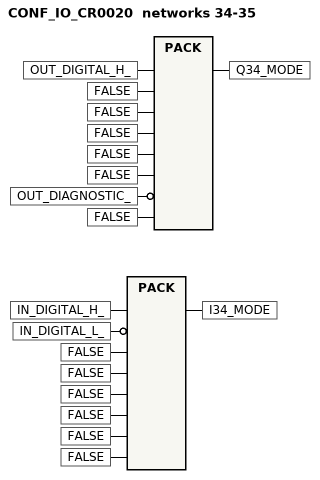
[picture p24: CONF_IO_CR0020 (FBD) networks 34-35]
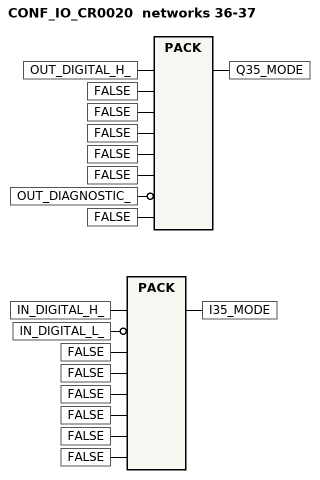
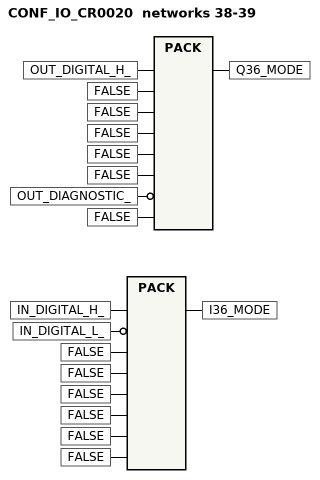
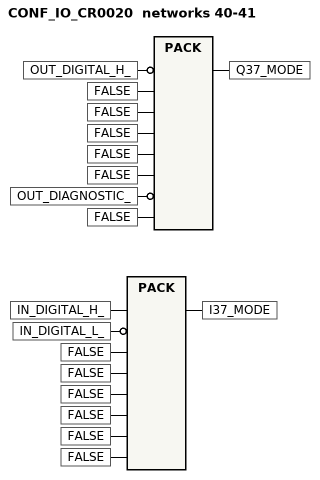
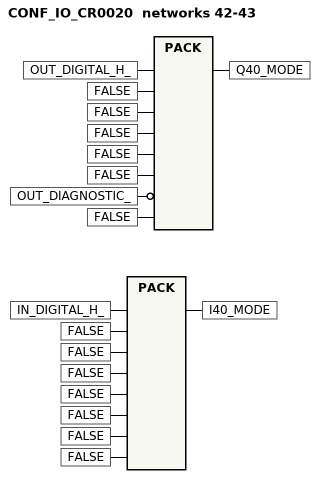
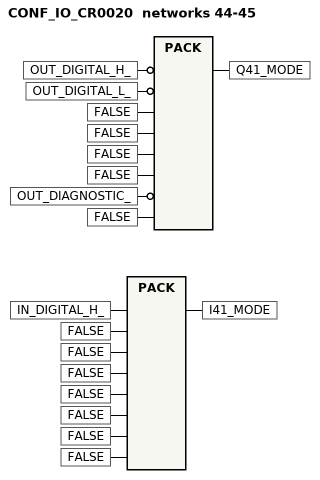
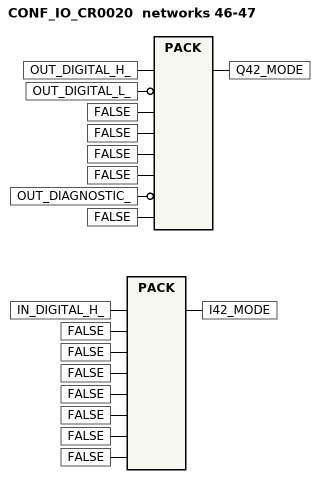
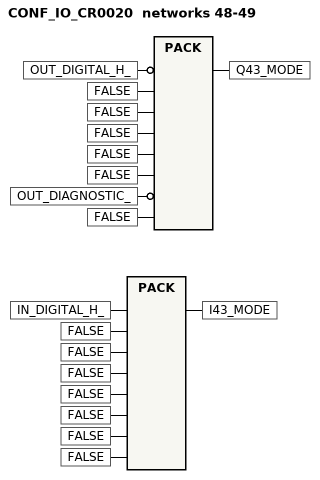
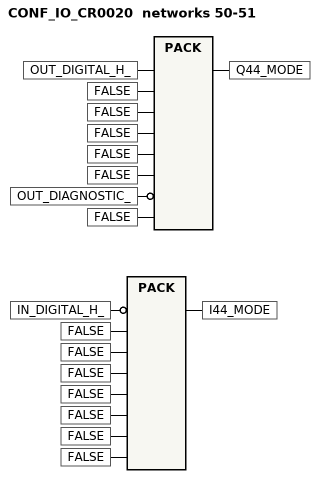
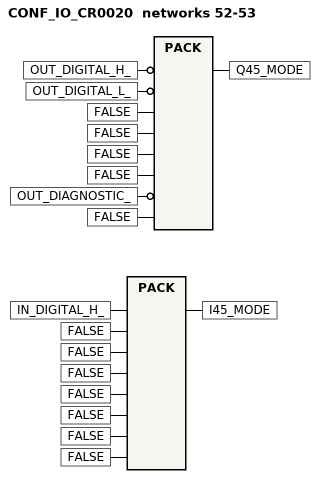
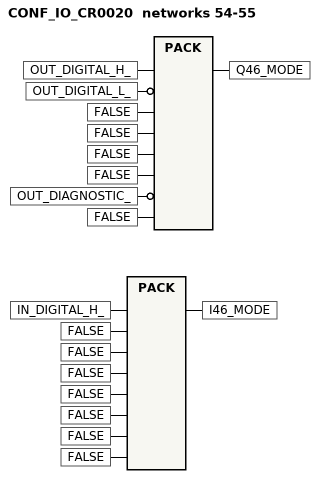
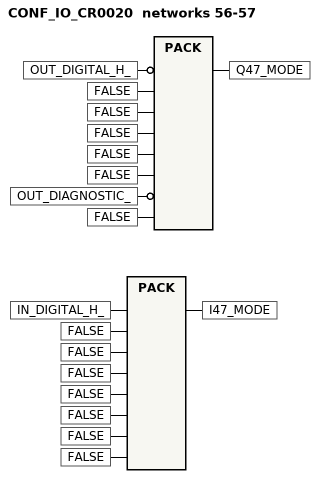
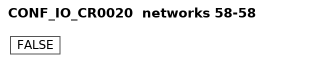
_FBD_ (* Function Block Diagram *)
NETWORK 1
	NOT INIT => >>END
NETWORK 2 (* Configuration byte for analog channel 0 pin 08 Connector 1. No output is connected to this pin. / Default setting:B0:=TRUE,B1:= FALSE,B2:= FALSE,B3:= FALSE,B4:= TRUE,B5:= FALSE,B6:= FALSE,B7:=FALSE *)
	PACK(FALSE, FALSE, IN_CURRENT_, FALSE, FALSE, FALSE, FALSE, FALSE) => I00_MODE
NETWORK 3 (* Configuration byte for analog channel 1 pin 27 Connector 1. No output is connected to this pin. / Default setting:B0:=TRUE,B1:= FALSE,B2:= FALSE,B3:= FALSE,B4:= TRUE,B5:= FALSE,B6:= FALSE,B7:=FALSE *)
	PACK(FALSE, FALSE, IN_CURRENT_, FALSE, FALSE, FALSE, FALSE, FALSE) => I01_MODE
NETWORK 4 (* Configuration byte for analog channel 2 pin 09 Connector 1. No output is connected to this pin. / Default setting:B0:=TRUE,B1:= FALSE,B2:= FALSE,B3:= FALSE,B4:= TRUE,B5:= FALSE,B6:= FALSE,B7:=FALSE *)
	PACK(FALSE, FALSE, IN_CURRENT_, FALSE, FALSE, FALSE, FALSE, FALSE) => I02_MODE
NETWORK 5 (* Configuration byte for analog channel 3 pin 28 Connector 1. No output is connected to this pin. / Default setting:B0:=TRUE,B1:= FALSE,B2:= FALSE,B3:= FALSE,B4:= TRUE,B5:= FALSE,B6:= FALSE,B7:=FALSE *)
	PACK(FALSE, FALSE, IN_CURRENT_, FALSE, FALSE, FALSE, FALSE, FALSE) => I03_MODE
NETWORK 6 (* Configuration byte for analog channel 4 pin 10 Connector 1. No output is connected to this pin. / Default setting:B0:=TRUE,B1:= FALSE,B2:= FALSE,B3:= FALSE,B4:= TRUE,B5:= FALSE,B6:= FALSE,B7:=FALSE *)
	PACK(FALSE, FALSE, IN_CURRENT_, FALSE, FALSE, FALSE, FALSE, FALSE) => I04_MODE
NETWORK 7 (* Configuration byte for analog channel 5 pin 29 Connector 1. No output is connected to this pin. / Default setting:B0:=TRUE,B1:= FALSE,B2:= FALSE,B3:= FALSE,B4:= TRUE,B5:= FALSE,B6:= FALSE,B7:=FALSE *)
	PACK(FALSE, FALSE, IN_CURRENT_, FALSE, FALSE, FALSE, FALSE, FALSE) => I05_MODE
NETWORK 8 (* Configuration byte for analog channel 6 pin 11 Connector 1. No output is connected to this pin. / Default setting:B0:=TRUE,B1:= FALSE,B2:= FALSE,B3:= FALSE,B4:= TRUE,B5:= FALSE,B6:= FALSE,B7:=FALSE *)
	PACK(FALSE, FALSE, IN_CURRENT_, FALSE, FALSE, FALSE, FALSE, FALSE) => I06_MODE
NETWORK 9 (* Configuration byte for analog channel 7 pin 30 Connector 1. No output is connected to this pin. / Default setting:B0:=TRUE,B1:= FALSE,B2:= FALSE,B3:= FALSE,B4:= TRUE,B5:= FALSE,B6:= FALSE,B7:=FALSE *)
	PACK(FALSE, FALSE, IN_CURRENT_, FALSE, FALSE, FALSE, FALSE, FALSE) => I07_MODE
NETWORK 10 (* Configuration byte for input %IX0.12  pin 20 Connector 1. No output is connected to this pin. / Default setting:B0:=TRUE,B1:= FALSE,B2:= FALSE,B3:= FALSE,B4:= FALSE,B5:= FALSE,B6:= FALSE,B7:=FALSE *)
	PACK(IN_DIGITAL_H_, FALSE, FALSE, FALSE, FALSE, FALSE, FALSE, NOT IN_FAST_) => I14_MODE
NETWORK 11 (* Configuration byte for input %IX0.13  pin 02 Connector 1. No output is connected to this pin. / Default setting:B0:=TRUE,B1:= FALSE,B2:= FALSE,B3:= FALSE,B4:= FALSE,B5:= FALSE,B6:= FALSE,B7:=FALSE *)
	PACK(IN_DIGITAL_H_, FALSE, FALSE, FALSE, FALSE, FALSE, FALSE, NOT IN_FAST_) => I15_MODE
NETWORK 12 (* Configuration byte for input %IX0.14  pin 21 Connector 1. No output is connected to this pin. / Default setting:B0:=TRUE,B1:= FALSE,B2:= FALSE,B3:= FALSE,B4:= FALSE,B5:= FALSE,B6:= FALSE,B7:=FALSE *)
	PACK(IN_DIGITAL_H_, FALSE, FALSE, FALSE, FALSE, FALSE, FALSE, IN_FAST_) => I16_MODE
NETWORK 13 (* Configuration byte for input %IX0.15  pin 38 Connector 1. No output is connected to this pin. / Default setting:B0:=TRUE,B1:= FALSE,B2:= FALSE,B3:= FALSE,B4:= FALSE,B5:= FALSE,B6:= FALSE,B7:=FALSE *)
	PACK(IN_DIGITAL_H_, FALSE, FALSE, FALSE, FALSE, FALSE, FALSE, IN_FAST_) => I17_MODE
NETWORK 14 (* Configuration byte for input %IX1.04  pin 19 Connector 1. No output is connected to this pin. / Default setting:B0:=TRUE,B1:= FALSE,B2:= FALSE,B3:= FALSE,B4:= FALSE,B5:= FALSE,B6:= FALSE,B7:=FALSE *)
	PACK(IN_DIGITAL_H_, FALSE, FALSE, FALSE, FALSE, FALSE, FALSE, IN_FAST_) => I24_MODE
NETWORK 15 (* Configuration byte for input %IX1.05  pin 55 Connector 1. No output is connected to this pin. / Default setting:B0:=TRUE,B1:= FALSE,B2:= FALSE,B3:= FALSE,B4:= FALSE,B5:= FALSE,B6:= FALSE,B7:=FALSE *)
	PACK(IN_DIGITAL_H_, FALSE, FALSE, FALSE, FALSE, FALSE, FALSE, IN_FAST_) => I25_MODE
NETWORK 16 (* Configuration byte for input %IX1.06  pin 18 Connector 1. No output is connected to this pin. / Default setting:B0:=TRUE,B1:= FALSE,B2:= FALSE,B3:= FALSE,B4:= FALSE,B5:= FALSE,B6:= FALSE,B7:=FALSE *)
	PACK(IN_DIGITAL_H_, FALSE, FALSE, FALSE, FALSE, FALSE, FALSE, IN_FAST_) => I26_MODE
NETWORK 17 (* Configuration byte for input %IX1.07  pin 37 Connector 1. No output is connected to this pin. / Default setting:B0:=TRUE,B1:= FALSE,B2:= FALSE,B3:= FALSE,B4:= FALSE,B5:= FALSE,B6:= FALSE,B7:=FALSE *)
	PACK(IN_DIGITAL_H_, FALSE, FALSE, FALSE, FALSE, FALSE, FALSE, IN_FAST_) => I27_MODE
NETWORK 18 (* Configuration byte for output %QX0.00  pin 44 Connector 1. The input %IX0.08 on pin 44 has no configuration byte. / Default setting:B0:=TRUE,B1:= FALSE,B2:= FALSE,B3:= FALSE,B4:= FALSE,B5:= FALSE,B6:= FALSE,B7:=TRUE *)
	PACK(OUT_DIGITAL_H_, FALSE, NOT OUT_CURRENT_, FALSE, FALSE, FALSE, NOT OUT_DIAGNOSTIC_, OUT_OVERLOAD_PROTECTION_) => Q10_MODE
NETWORK 19 (* Configuration byte for output %QX0.01  pin 45 Connector 1. The input %IX0.09 on pin 45 has no configuration byte. / Default setting:B0:=TRUE,B1:= FALSE,B2:= FALSE,B3:= FALSE,B4:= FALSE,B5:= FALSE,B6:= FALSE,B7:=TRUE *)
	PACK(OUT_DIGITAL_H_, FALSE, NOT OUT_CURRENT_, FALSE, FALSE, FALSE, NOT OUT_DIAGNOSTIC_, OUT_OVERLOAD_PROTECTION_) => Q11_MODE
NETWORK 20 (* Configuration byte for output %QX0.02  pin 46 Connector 1. The input %IX0.10 on pin 46 has no configuration byte. / Default setting:B0:=TRUE,B1:= FALSE,B2:= FALSE,B3:= FALSE,B4:= FALSE,B5:= FALSE,B6:= FALSE,B7:=TRUE *)
	PACK(OUT_DIGITAL_H_, FALSE, NOT OUT_CURRENT_, FALSE, FALSE, FALSE, NOT OUT_DIAGNOSTIC_, OUT_OVERLOAD_PROTECTION_) => Q12_MODE
NETWORK 21 (* Configuration byte for output %QX0.03  pin 47 Connector 1. The input %IX0.11 on pin 47 has no configuration byte. / Default setting:B0:=TRUE,B1:= FALSE,B2:= FALSE,B3:= FALSE,B4:= FALSE,B5:= FALSE,B6:= FALSE,B7:=TRUE *)
	PACK(OUT_DIGITAL_H_, FALSE, NOT OUT_CURRENT_, FALSE, FALSE, FALSE, NOT OUT_DIAGNOSTIC_, OUT_OVERLOAD_PROTECTION_) => Q13_MODE
NETWORK 22 (* Configuration byte for output %QX0.04  pin 36 Connector 1. The input %IX1.00 on pin 36 has no configuration byte. / Default setting:B0:=TRUE,B1:= FALSE,B2:= FALSE,B3:= FALSE,B4:= FALSE,B5:= FALSE,B6:= FALSE,B7:=TRUE *)
	PACK(OUT_DIGITAL_H_, FALSE, NOT OUT_CURRENT_, FALSE, FALSE, FALSE, NOT OUT_DIAGNOSTIC_, OUT_OVERLOAD_PROTECTION_) => Q20_MODE
NETWORK 23 (* Configuration byte for output %QX0.05  pin 54 Connector 1 The input %IX1.01 on pin 54 has no configuration byte. / Default setting:B0:=TRUE,B1:= FALSE,B2:= FALSE,B3:= FALSE,B4:= FALSE,B5:= FALSE,B6:= FALSE,B7:=TRUE *)
	PACK(OUT_DIGITAL_H_, FALSE, NOT OUT_CURRENT_, FALSE, FALSE, FALSE, NOT OUT_DIAGNOSTIC_, OUT_OVERLOAD_PROTECTION_) => Q21_MODE
NETWORK 24 (* Configuration byte for output %QX0.06  pin 17 Connector 1 The input %IX1.02 on pin 17 has no configuration byte. / Default setting:B0:=TRUE,B1:= FALSE,B2:= FALSE,B3:= FALSE,B4:= FALSE,B5:= FALSE,B6:= FALSE,B7:=TRUE *)
	PACK(NOT OUT_DIGITAL_H_, FALSE, NOT OUT_CURRENT_, FALSE, FALSE, FALSE, NOT OUT_DIAGNOSTIC_, OUT_OVERLOAD_PROTECTION_) => Q22_MODE
NETWORK 25 (* Configuration byte for output %QX0.07  pin 53 Connector 1 The input %IX1.03 on pin 53 has no configuration byte. / Default setting:B0:=TRUE,B1:= FALSE,B2:= FALSE,B3:= FALSE,B4:= FALSE,B5:= FALSE,B6:= FALSE,B7:=TRUE *)
	PACK(OUT_DIGITAL_H_, FALSE, NOT OUT_CURRENT_, FALSE, FALSE, FALSE, NOT OUT_DIAGNOSTIC_, OUT_OVERLOAD_PROTECTION_) => Q23_MODE
NETWORK 26 (* Configuration byte for output %QX0.08  pin 39 Connector 1. / Default setting:B0:=TRUE,B1:= FALSE,B2:= FALSE,B3:= FALSE,B4:= FALSE,B5:= FALSE,B6:= FALSE,B7:=FALSE *)
	PACK(NOT OUT_DIGITAL_H_, FALSE, FALSE, FALSE, FALSE, FALSE, NOT OUT_DIAGNOSTIC_, FALSE) => Q30_MODE
NETWORK 27 (* Configuration byte for input %IX1.08  pin 39 Connector 1. / Default setting:B0:=TRUE,B1:= FALSE,B2:= FALSE,B3:= FALSE,B4:= FALSE,B5:= FALSE,B6:= FALSE,B7:=FALSE *)
	PACK(IN_DIGITAL_H_, NOT IN_DIGITAL_L_, FALSE, FALSE, FALSE, FALSE, FALSE, FALSE) => I30_MODE
NETWORK 28 (* Configuration byte for output %QX0.09  pin 03 Connector 1. / Default setting:B0:=TRUE,B1:= FALSE,B2:= FALSE,B3:= FALSE,B4:= FALSE,B5:= FALSE,B6:= FALSE,B7:=FALSE *)
	PACK(NOT OUT_DIGITAL_H_, FALSE, FALSE, FALSE, FALSE, FALSE, NOT OUT_DIAGNOSTIC_, FALSE) => Q31_MODE
NETWORK 29 (* Configuration byte for input %IX1.09  pin 03 Connector 1. / Default setting:B0:=TRUE,B1:= FALSE,B2:= FALSE,B3:= FALSE,B4:= FALSE,B5:= FALSE,B6:= FALSE,B7:=FALSE *)
	PACK(IN_DIGITAL_H_, NOT IN_DIGITAL_L_, FALSE, FALSE, FALSE, FALSE, FALSE, FALSE) => I31_MODE
NETWORK 30 (* Configuration byte for output %QX0.10  pin 40 Connector 1. / Default setting:B0:=TRUE,B1:= FALSE,B2:= FALSE,B3:= FALSE,B4:= FALSE,B5:= FALSE,B6:= FALSE,B7:=FALSE *)
	PACK(NOT OUT_DIGITAL_H_, FALSE, FALSE, FALSE, FALSE, FALSE, NOT OUT_DIAGNOSTIC_, FALSE) => Q32_MODE
NETWORK 31 (* Configuration byte forintput %IX1.10  pin 40 Connector 1. / Default setting:B0:=TRUE,B1:= FALSE,B2:= FALSE,B3:= FALSE,B4:= FALSE,B5:= FALSE,B6:= FALSE,B7:=FALSE *)
	PACK(IN_DIGITAL_H_, NOT IN_DIGITAL_L_, FALSE, FALSE, FALSE, FALSE, FALSE, FALSE) => I32_MODE
NETWORK 32 (* Configuration byte for output %QX0.11  pin 22 Connector 1. / Default setting:B0:=TRUE,B1:= FALSE,B2:= FALSE,B3:= FALSE,B4:= FALSE,B5:= FALSE,B6:= FALSE,B7:=FALSE *)
	PACK(OUT_DIGITAL_H_, FALSE, FALSE, FALSE, FALSE, FALSE, NOT OUT_DIAGNOSTIC_, FALSE) => Q33_MODE
NETWORK 33 (* Configuration byte for input %IX1.11  pin 22 Connector 1. / Default setting:B0:=TRUE,B1:= FALSE,B2:= FALSE,B3:= FALSE,B4:= FALSE,B5:= FALSE,B6:= FALSE,B7:=FALSE *)
	PACK(IN_DIGITAL_H_, NOT IN_DIGITAL_L_, FALSE, FALSE, FALSE, FALSE, FALSE, FALSE) => I33_MODE
NETWORK 34 (* Configuration byte for output %QX0.12  pin 41 Connector 1. / Default setting:B0:=TRUE,B1:= FALSE,B2:= FALSE,B3:= FALSE,B4:= FALSE,B5:= FALSE,B6:= FALSE,B7:=FALSE *)
	PACK(OUT_DIGITAL_H_, FALSE, FALSE, FALSE, FALSE, FALSE, NOT OUT_DIAGNOSTIC_, FALSE) => Q34_MODE
NETWORK 35 (* Configuration byte for input %IX1.12  pin 41 Connector 1. / Default setting:B0:=TRUE,B1:= FALSE,B2:= FALSE,B3:= FALSE,B4:= FALSE,B5:= FALSE,B6:= FALSE,B7:=FALSE *)
	PACK(IN_DIGITAL_H_, NOT IN_DIGITAL_L_, FALSE, FALSE, FALSE, FALSE, FALSE, FALSE) => I34_MODE
NETWORK 36 (* Configuration byte for output %QX0.13  pin 42 Connector 1. / Default setting:B0:=TRUE,B1:= FALSE,B2:= FALSE,B3:= FALSE,B4:= FALSE,B5:= FALSE,B6:= FALSE,B7:=FALSE *)
	PACK(OUT_DIGITAL_H_, FALSE, FALSE, FALSE, FALSE, FALSE, NOT OUT_DIAGNOSTIC_, FALSE) => Q35_MODE
NETWORK 37 (* Configuration byte for input %IX1.13  pin 42 Connector 1. / Default setting:B0:=TRUE,B1:= FALSE,B2:= FALSE,B3:= FALSE,B4:= FALSE,B5:= FALSE,B6:= FALSE,B7:=FALSE *)
	PACK(IN_DIGITAL_H_, NOT IN_DIGITAL_L_, FALSE, FALSE, FALSE, FALSE, FALSE, FALSE) => I35_MODE
NETWORK 38 (* Configuration byte for output %QX0.14  pin 43 Connector 1. / Default setting:B0:=TRUE,B1:= FALSE,B2:= FALSE,B3:= FALSE,B4:= FALSE,B5:= FALSE,B6:= FALSE,B7:=FALSE *)
	PACK(OUT_DIGITAL_H_, FALSE, FALSE, FALSE, FALSE, FALSE, NOT OUT_DIAGNOSTIC_, FALSE) => Q36_MODE
NETWORK 39 (* Configuration byte for input %IX1.14  pin 43 Connector 1. / Default setting:B0:=TRUE,B1:= FALSE,B2:= FALSE,B3:= FALSE,B4:= FALSE,B5:= FALSE,B6:= FALSE,B7:=FALSE *)
	PACK(IN_DIGITAL_H_, NOT IN_DIGITAL_L_, FALSE, FALSE, FALSE, FALSE, FALSE, FALSE) => I36_MODE
NETWORK 40 (* Configuration byte for output %QX0.15  pin 04 Connector 1. / Default setting:B0:=TRUE,B1:= FALSE,B2:= FALSE,B3:= FALSE,B4:= FALSE,B5:= FALSE,B6:= FALSE,B7:=FALSE *)
	PACK(NOT OUT_DIGITAL_H_, FALSE, FALSE, FALSE, FALSE, FALSE, NOT OUT_DIAGNOSTIC_, FALSE) => Q37_MODE
NETWORK 41 (* Configuration byte for input %IX1.15  pin 04 Connector 1. / Default setting:B0:=TRUE,B1:= FALSE,B2:= FALSE,B3:= FALSE,B4:= FALSE,B5:= FALSE,B6:= FALSE,B7:=FALSE *)
	PACK(IN_DIGITAL_H_, NOT IN_DIGITAL_L_, FALSE, FALSE, FALSE, FALSE, FALSE, FALSE) => I37_MODE
NETWORK 42 (* Configuration byte for output %QX1.00  pin 48 Connector 1. / Default setting:B0:=FALSE,B1:= FALSE,B2:= FALSE,B3:= FALSE,B4:= FALSE,B5:= FALSE,B6:= FALSE,B7:=FALSE *)
	PACK(OUT_DIGITAL_H_, FALSE, FALSE, FALSE, FALSE, FALSE, NOT OUT_DIAGNOSTIC_, FALSE) => Q40_MODE
NETWORK 43 (* Configuration byte for intput %IX2.00  pin 48 Connector 1. / Default setting:B0:=TRUE,B1:= FALSE,B2:= FALSE,B3:= FALSE,B4:= FALSE,B5:= FALSE,B6:= FALSE,B7:=FALSE *)
	PACK(IN_DIGITAL_H_, FALSE, FALSE, FALSE, FALSE, FALSE, FALSE, FALSE) => I40_MODE
NETWORK 44 (* Configuration byte for output %QX1.01  pin 49 Connector 1. / Default setting:B0:=FALSE,B1:= FALSE,B2:= FALSE,B3:= FALSE,B4:= FALSE,B5:= FALSE,B6:= FALSE,B7:=FALSE *)
	PACK(NOT OUT_DIGITAL_H_, NOT OUT_DIGITAL_L_, FALSE, FALSE, FALSE, FALSE, NOT OUT_DIAGNOSTIC_, FALSE) => Q41_MODE
NETWORK 45 (* Configuration byte for input %IX2.01  pin 49 Connector 1. / Default setting:B0:=TRUE,B1:= FALSE,B2:= FALSE,B3:= FALSE,B4:= FALSE,B5:= FALSE,B6:= FALSE,B7:=FALSE *)
	PACK(IN_DIGITAL_H_, FALSE, FALSE, FALSE, FALSE, FALSE, FALSE, FALSE) => I41_MODE
NETWORK 46 (* Configuration byte for output %QX1.02  pin 31 Connector 1. / Default setting:B0:=FALSE,B1:= FALSE,B2:= FALSE,B3:= FALSE,B4:= FALSE,B5:= FALSE,B6:= FALSE,B7:=FALSE *)
	PACK(OUT_DIGITAL_H_, NOT OUT_DIGITAL_L_, FALSE, FALSE, FALSE, FALSE, NOT OUT_DIAGNOSTIC_, FALSE) => Q42_MODE
NETWORK 47 (* Configuration byte for input %IX2.02  pin 31 Connector 1. / Default setting:B0:=TRUE,B1:= FALSE,B2:= FALSE,B3:= FALSE,B4:= FALSE,B5:= FALSE,B6:= FALSE,B7:=FALSE *)
	PACK(IN_DIGITAL_H_, FALSE, FALSE, FALSE, FALSE, FALSE, FALSE, FALSE) => I42_MODE
NETWORK 48 (* Configuration byte for output %QX1.03  pin 50 Connector 1. / Default setting:B0:=FALSE,B1:= FALSE,B2:= FALSE,B3:= FALSE,B4:= FALSE,B5:= FALSE,B6:= FALSE,B7:=FALSE *)
	PACK(NOT OUT_DIGITAL_H_, FALSE, FALSE, FALSE, FALSE, FALSE, NOT OUT_DIAGNOSTIC_, FALSE) => Q43_MODE
NETWORK 49 (* Configuration byte for input %IX2.03  pin 50 Connector 1. / Default setting:B0:=TRUE,B1:= FALSE,B2:= FALSE,B3:= FALSE,B4:= FALSE,B5:= FALSE,B6:= FALSE,B7:=FALSE *)
	PACK(IN_DIGITAL_H_, FALSE, FALSE, FALSE, FALSE, FALSE, FALSE, FALSE) => I43_MODE
NETWORK 50 (* Configuration byte for output %QX1.04  pin 51 Connector 1. / Default setting:B0:=FALSE,B1:= FALSE,B2:= FALSE,B3:= FALSE,B4:= FALSE,B5:= FALSE,B6:= FALSE,B7:=FALSE *)
	PACK(OUT_DIGITAL_H_, FALSE, FALSE, FALSE, FALSE, FALSE, NOT OUT_DIAGNOSTIC_, FALSE) => Q44_MODE
NETWORK 51 (* Configuration byte for input %IX2.04  pin 51 Connector 1. / Default setting:B0:=TRUE,B1:= FALSE,B2:= FALSE,B3:= FALSE,B4:= FALSE,B5:= FALSE,B6:= FALSE,B7:=FALSE *)
	PACK(NOT IN_DIGITAL_H_, FALSE, FALSE, FALSE, FALSE, FALSE, FALSE, FALSE) => I44_MODE
NETWORK 52 (* Configuration byte for output %QX1.05  pin 52 Connector 1. / Default setting:B0:=FALSE,B1:= FALSE,B2:= FALSE,B3:= FALSE,B4:= FALSE,B5:= FALSE,B6:= FALSE,B7:=FALSE *)
	PACK(NOT OUT_DIGITAL_H_, NOT OUT_DIGITAL_L_, FALSE, FALSE, FALSE, FALSE, NOT OUT_DIAGNOSTIC_, FALSE) => Q45_MODE
NETWORK 53 (* Configuration byte for input %IX1.05  pin 52 Connector 1. / Default setting:B0:=TRUE,B1:= FALSE,B2:= FALSE,B3:= FALSE,B4:= FALSE,B5:= FALSE,B6:= FALSE,B7:=FALSE *)
	PACK(IN_DIGITAL_H_, FALSE, FALSE, FALSE, FALSE, FALSE, FALSE, FALSE) => I45_MODE
NETWORK 54 (* Configuration byte for output %QX1.06  pin 16 Connector 1. / Default setting:B0:=FALSE,B1:= FALSE,B2:= FALSE,B3:= FALSE,B4:= FALSE,B5:= FALSE,B6:= FALSE,B7:=FALSE *)
	PACK(OUT_DIGITAL_H_, NOT OUT_DIGITAL_L_, FALSE, FALSE, FALSE, FALSE, NOT OUT_DIAGNOSTIC_, FALSE) => Q46_MODE
NETWORK 55 (* Configuration byte for input %IX2.06  pin 16 Connector 1. / Default setting:B0:=TRUE,B1:= FALSE,B2:= FALSE,B3:= FALSE,B4:= FALSE,B5:= FALSE,B6:= FALSE,B7:=FALSE *)
	PACK(IN_DIGITAL_H_, FALSE, FALSE, FALSE, FALSE, FALSE, FALSE, FALSE) => I46_MODE
NETWORK 56 (* Configuration byte for output %QX1.07  pin 35 Connector 1. / Default setting:B0:=FALSE,B1:= FALSE,B2:= FALSE,B3:= FALSE,B4:= FALSE,B5:= FALSE,B6:= FALSE,B7:=FALSE *)
	PACK(NOT OUT_DIGITAL_H_, FALSE, FALSE, FALSE, FALSE, FALSE, NOT OUT_DIAGNOSTIC_, FALSE) => Q47_MODE
NETWORK 57 (* Configuration byte for input %IX2.07  pin 35 Connector 1. / Default setting:B0:=TRUE,B1:= FALSE,B2:= FALSE,B3:= FALSE,B4:= FALSE,B5:= FALSE,B6:= FALSE,B7:=FALSE *)
	PACK(IN_DIGITAL_H_, FALSE, FALSE, FALSE, FALSE, FALSE, FALSE, FALSE) => I47_MODE
NETWORK 58 END::
	FALSE
_END_FBD_
END_PROGRAM

(* POU PLC_CYCLE, ST *)
PROGRAM PLC_CYCLE

VAR
	old_cycle           : DWORD;
	TIMER_READ_US1      : TIMER_READ_US;
	cycle               : DWORD;
	init                : BOOL := 1;
END_VAR

VAR_OUTPUT
	cycletime_us        : DWORD;
	max_cycle_us        : DWORD;
END_VAR

VAR_INPUT
	reset_max_cycletime : BOOL;
END_VAR
(*-----------------------------------------------------------------------------------------------------------------------------------------------------------------------------------*)
(**)

TIMER_READ_US1(TIME_US => cycle );
cycletime_us := cycle - old_cycle;
old_cycle := cycle;

IF max_cycle_us < cycletime_us AND NOT init THEN
	max_cycle_us := cycletime_us;
END_IF;

IF reset_max_cycletime THEN
	max_cycle_us := 0;
END_IF;

init := 0;
END_PROGRAM

(* POU Service/CRC_processing, ST *)
PROGRAM CRC_processing

VAR_INPUT
	bInit      : BOOL;
END_VAR

VAR
	CHECK_DATA : CHECK_DATA;
END_VAR
(*CHECK_DATA(STARTADR := 50_000, LENGTH := 100, UPDATE := bInit, RESULT => , CHECKSUM => );*)

dwMS_ProgramCRC := 1357924680;
END_PROGRAM

(* POU Service/ID_Program_processing, ST *)
PROGRAM ID_Program_processing

VAR_INPUT
	bInit               : BOOL;
END_VAR

VAR
	(*byNumVersion        : BYTE := 4;(*Номер версии (соответствует типу установки)*)*)
	(*byNumCorrection     : BYTE := 0;(*Номер исправления*)*)
	(*iNumOrder           : INT  := 593;(*Номер заказа*)*)
	byDeviceTypeAppType : BYTE;

	bECU1_CurrentStat_1 : BYTE;
	bECU1_CurrentStat_2 : BYTE;

	bECU2_CurrentStat_1 : BYTE;
	bECU2_CurrentStat_2 : BYTE;

	instMemCpy          : MEMCPY;
END_VAR
(*-----------------------------------------------------------------------------------------------------------------------------------------------------------------------------------*)
(**)

(*instMemCpy(DST := ADR(abyMS_ProgramID[0]), SRC := ADR(iNumOrder),       LEN := 2);*)
(*instMemCpy(DST := ADR(abyMS_ProgramID[2]), SRC := ADR(byNumCorrection), LEN := 1);*)
(*instMemCpy(DST := ADR(abyMS_ProgramID[3]), SRC := ADR(byNumVersion),    LEN := 1);*)

byDeviceTypeAppType := 16#00;

byDeviceTypeAppType := byUnitTypePrimaryApp OR SHL(byProgrammableDeviceType, 4);

instMemCpy(DST := ADR(abyMS_ProgramID[0]), SRC := ADR(byFixNumber),                  LEN := 1);
instMemCpy(DST := ADR(abyMS_ProgramID[1]), SRC := ADR(byUnitModificationPrimaryApp), LEN := 1);
instMemCpy(DST := ADR(abyMS_ProgramID[2]), SRC := ADR(byUnitModelPrimaryApp),        LEN := 1);
instMemCpy(DST := ADR(abyMS_ProgramID[3]), SRC := ADR(byDeviceTypeAppType),          LEN := 1);

bECU1_CurrentStat_1:=PACK(B0:=ERROR,
							B1:=CLAMP_15,
							B2:=ERROR_MEMORY,
							B3:=ERROR_TEMPERATURE,
							B4:=ERROR_VBBR,
							B5:=RELAY_CLAMP_15,
							B6:=RELAIS,
							B7:=ERROR_POWER);(*Собираем 1-й байт состояния контроллера #1*)

bECU1_CurrentStat_2:=PACK(B0:=TEST,
							B1:=FALSE,
							B2:=FALSE,
							B3:=FALSE,
							B4:=FALSE,
							B5:=FALSE,
							B6:=FALSE,
							B7:=FALSE);(*Собираем 2-й байт состояния контроллера #1*)

bECU2_CurrentStat_1:=PACK(B0:=FALSE,
							B1:=FALSE,
							B2:=FALSE,
							B3:=FALSE,
							B4:=FALSE,
							B5:=FALSE,
							B6:=FALSE,
							B7:=FALSE);(*Собираем 1-й байт состояния контроллера #2*)

bECU2_CurrentStat_2:=PACK(B0:=FALSE,
							B1:=FALSE,
							B2:=FALSE,
							B3:=FALSE,
							B4:=FALSE,
							B5:=FALSE,
							B6:=FALSE,
							B7:=FALSE);(*Собираем 2-й байт состояния контроллера #2*)

instMemCpy(DST:=ADR(abyDataStateMS[0]),  SRC:=ADR(bECU1_CurrentStat_1), LEN:=1);
instMemCpy(DST:=ADR(abyDataStateMS[1]),  SRC:=ADR(bECU1_CurrentStat_2), LEN:=1);
instMemCpy(DST:=ADR(abyDataStateSL1[0]), SRC:=ADR(bECU2_CurrentStat_1), LEN:=1);
instMemCpy(DST:=ADR(abyDataStateSL1[1]), SRC:=ADR(bECU2_CurrentStat_2), LEN:=1);

rECU_SupplyVoltage := WORD_TO_REAL(SUPPLY_VOLTAGE) / 10;
rECU_Temperature   := -9999;
END_PROGRAM

(* POU Service/Time_processing, ST *)
PROGRAM Time_processing

VAR
	TIMER_READ_US1 : TIMER_READ_US;
END_VAR
(*-----------------------------------------------------------------------------------------------------------------------------------------------------------------------------------*)
(**)

TIMER_READ_US1(TIME_US => dwTime_US);
END_PROGRAM

(* POU Service/Timer_processing, ST *)
PROGRAM Timer_processing

VAR_INPUT
	bFirstIn   : BOOL;
END_VAR

VAR
	TPInstHigh : TP;
	TPInstLow  : TP;
END_VAR
(*-----------------------------------------------------------------------------------------------------------------------------------------------------------------------------------*)
(*Формируем импульсы для управления лампочками*)

TPInstHigh(IN := NOT TPInstLow.Q, PT := T#0.25s, Q => bTimerBlinkOut, ET => );

TPInstLow(IN := NOT TPInstHigh.Q, PT := T#0.25s, Q => , ET => );
END_PROGRAM

(* POU Default_Settings/First_Start_processing, ST *)
PROGRAM First_Start_processing

VAR
	dwFirstStartIdMemo   : DWORD;
	dwFirstStartIdCode   : DWORD := 06031979;
	dwFirstStartCurrMode : DWORD := 1;
	instFRAMWrite        : FRAMWRITE;
	instFRAMRead         : FRAMREAD;
	i                    : INT;
END_VAR
(*-----------------------------------------------------------------------------------------------------------------------------------------------------------------------------------*)
(*Читаем идентификатор наличия предыдущей программы*)

instFRAMRead(Enable := 1, SRC := iMemAdrFirstStartId, LEN := 4, DST := ADR(dwFirstStartIdMemo));(*Читаем идентификатор наличия предыдущей программы*)

IF dwFirstStartIdMemo <> dwFirstStartIdCode
THEN

(*

FOR i := 0 TO iSizeArrayParamMax - 1 DO
	dwArrayParam00[i] := 16#FFFF;
	instFRAMWrite(Enable := TRUE, DST := iMemAdrArrayParam00 + (i - 1) * 4, LEN := 4, SRC := ADR(dwArrayParam00[i]));(**)
END_FOR;

(*Запись в FRAM коэффициентов для каналов АЦП*)
	FOR i := 1 TO 16 DO
		instFRAMWrite(Enable := TRUE, DST := iMemAdrArrayParam01 + (i - 1) * 4, LEN := 4, SRC := ADR(rArrayDataADC_XH[i]));(*Запись в FRAM заводской установки MAX шкалы текущего канала*)
		instFRAMWrite(Enable := TRUE, DST := iMemAdrArrayParam02 + (i - 1) * 4, LEN := 4, SRC := ADR(rArrayDataADC_XL[i]));(*Запись в FRAM заводской установки MIN шкалы текущего канала*)
	END_FOR;

*)

(*Устанавливаем стартовый режим*)
	instFRAMWrite(Enable := 1, DST := iMemAdrCurrMode, LEN := 4, SRC := ADR(dwFirstStartCurrMode));(*Записываем идентификатор режима "Работа"*)
	bCurrModeChange := 1;

	instFRAMWrite(Enable := 1, DST := iMemAdrFirstStartId, LEN := 4, SRC := ADR(dwFirstStartIdCode));(*Записываем идентификатор наличия предыдущей программы*)

END_IF;
END_PROGRAM

(* POU CAN1_J1939/CAN1_J1939_Setting, ST *)
PROGRAM CAN1_J1939_Setting

VAR_INPUT
	bInit      : BOOL;
END_VAR

VAR
	CAN1_SET   : CAN1_EXT;
	CAN1_J1939 : J1939_1;
END_VAR
(*-----------------------------------------------------------------------------------------------------------------------------------------------------------------------------------*)
(**)

CAN1_SET(ENABLE := bCAN1_TransmitEnable, START := bInit, EXTENDED_MODE := 1,  BAUDRATE := wCAN1_BaudRate);
CAN1_J1939(ENABLE := bCAN1_TransmitEnable, START := bInit, MY_ADDRESS := byCAN1_PreferAddr);
END_PROGRAM

(* POU CAN2_J1939/CAN2_J1939_Setting, ST *)
PROGRAM CAN2_J1939_Setting

VAR_INPUT
	bInit      : BOOL;
END_VAR

VAR
	CAN2_SET   : CAN2;
	CAN2_J1939 : J1939_2;
END_VAR
(*-----------------------------------------------------------------------------------------------------------------------------------------------------------------------------------*)
(**)

CAN2_SET(ENABLE := bCAN2_TransmitEnable, START := bInit, EXTENDED_MODE := 1,  BAUDRATE := wCAN2_BaudRate);
CAN2_J1939(ENABLE := bCAN2_TransmitEnable, START := bInit, MY_ADDRESS := byCAN2_PreferAddr);
END_PROGRAM

(* POU CAN1_J1939/CAN1_J1939_Receive_processing, ST *)
PROGRAM CAN1_J1939_Receive_processing

VAR_INPUT
	bInit                         : BOOL;
END_VAR

VAR
	dwControlCAN1RX_CHANNEL_INDEX : DWORD;
	dwControlCAN1RX_PARAM00       : DWORD;
	dwControlCAN1RX_PARAM09       : DWORD;
	bControlCAN1RX_CHANNEL_INDEX  : BOOL;
	bControlCAN1RX_PARAM00        : BOOL;
	bControlCAN1RX_PARAM09        : BOOL;

	instFRAMWrite                 : FRAMWRITE;
	instMemCpy                    : MEMCPY;
END_VAR
(*-----------------------------------------------------------------------------------------------------------------------------------------------------------------------------------*)
(**)

bCommand:=0;(*Сброс флага "Получена новая команда"*)

(*-----------------------------------------------------------------------------------------------------------------------------------------------------------------------------------*)
(*Принимаем сообщения CAN J1939*)

  CAN1RX_UNIT_ADDR     (ENABLE := 1, CONFIG := bInit, PG := 0, PF := PGN_TO_PF(dwPGN1_UNIT_ADDR),     PS := PGN_TO_PS(dwPGN1_UNIT_ADDR),     DST := ADR(abyCAN1RX_UNIT_ADDR),     RPT := T#0S, LIFE := , RESULT => , DEVICE => , LEN => );

  CAN1RX_CHANNEL_INDEX (ENABLE := 1, CONFIG := bInit, PG := 0, PF := PGN_TO_PF(dwPGN1_CHANNEL_INDEX), PS := PGN_TO_PS(dwPGN1_CHANNEL_INDEX), DST := ADR(abyCAN1RX_CHANNEL_INDEX), RPT := T#0S, LIFE := , RESULT => , DEVICE => , LEN => );
  CAN1RX_PARAM00       (ENABLE := 1, CONFIG := bInit, PG := 0, PF := PGN_TO_PF(dwPGN1_PARAM00),       PS := PGN_TO_PS(dwPGN1_PARAM00),       DST := ADR(abyCAN1RX_PARAM00),       RPT := T#0S, LIFE := , RESULT => , DEVICE => , LEN => );
  CAN1RX_PARAM01       (ENABLE := 1, CONFIG := bInit, PG := 0, PF := PGN_TO_PF(dwPGN1_PARAM01),       PS := PGN_TO_PS(dwPGN1_PARAM01),       DST := ADR(abyCAN1RX_PARAM01),       RPT := T#0S, LIFE := , RESULT => , DEVICE => , LEN => );
  CAN1RX_PARAM02       (ENABLE := 1, CONFIG := bInit, PG := 0, PF := PGN_TO_PF(dwPGN1_PARAM02),       PS := PGN_TO_PS(dwPGN1_PARAM02),       DST := ADR(abyCAN1RX_PARAM02),       RPT := T#0S, LIFE := , RESULT => , DEVICE => , LEN => );
  CAN1RX_PARAM03       (ENABLE := 1, CONFIG := bInit, PG := 0, PF := PGN_TO_PF(dwPGN1_PARAM03),       PS := PGN_TO_PS(dwPGN1_PARAM03),       DST := ADR(abyCAN1RX_PARAM03),       RPT := T#0S, LIFE := , RESULT => , DEVICE => , LEN => );
  CAN1RX_PARAM04       (ENABLE := 1, CONFIG := bInit, PG := 0, PF := PGN_TO_PF(dwPGN1_PARAM04),       PS := PGN_TO_PS(dwPGN1_PARAM04),       DST := ADR(abyCAN1RX_PARAM04),       RPT := T#0S, LIFE := , RESULT => , DEVICE => , LEN => );
  CAN1RX_PARAM05       (ENABLE := 1, CONFIG := bInit, PG := 0, PF := PGN_TO_PF(dwPGN1_PARAM05),       PS := PGN_TO_PS(dwPGN1_PARAM05),       DST := ADR(abyCAN1RX_PARAM05),       RPT := T#0S, LIFE := , RESULT => , DEVICE => , LEN => );
  CAN1RX_PARAM06       (ENABLE := 1, CONFIG := bInit, PG := 0, PF := PGN_TO_PF(dwPGN1_PARAM06),       PS := PGN_TO_PS(dwPGN1_PARAM06),       DST := ADR(abyCAN1RX_PARAM06),       RPT := T#0S, LIFE := , RESULT => , DEVICE => , LEN => );
  CAN1RX_PARAM07       (ENABLE := 1, CONFIG := bInit, PG := 0, PF := PGN_TO_PF(dwPGN1_PARAM07),       PS := PGN_TO_PS(dwPGN1_PARAM07),       DST := ADR(abyCAN1RX_PARAM07),       RPT := T#0S, LIFE := , RESULT => , DEVICE => , LEN => );
(*CAN1RX_PARAM08       (ENABLE := 1, CONFIG := bInit, PG := 0, PF := PGN_TO_PF(dwPGN1_PARAM08),       PS := PGN_TO_PS(dwPGN1_PARAM08),       DST := ADR(abyCAN1RX_PARAM08),       RPT := T#0S, LIFE := , RESULT => , DEVICE => , LEN => );*)
  CAN1RX_PARAM09       (ENABLE := 1, CONFIG := bInit, PG := 0, PF := PGN_TO_PF(dwPGN1_PARAM09),       PS := PGN_TO_PS(dwPGN1_PARAM09),       DST := ADR(abyCAN1RX_PARAM09),       RPT := T#0S, LIFE := , RESULT => , DEVICE => , LEN => );
  CAN1RX_PARAM10       (ENABLE := 1, CONFIG := bInit, PG := 0, PF := PGN_TO_PF(dwPGN1_PARAM10),       PS := PGN_TO_PS(dwPGN1_PARAM10),       DST := ADR(abyCAN1RX_PARAM10),       RPT := T#0S, LIFE := , RESULT => , DEVICE => , LEN => );

  CAN1RX_CURR_MODE     (ENABLE := 1, CONFIG := bInit, PG := 0, PF := PGN_TO_PF(dwPGN1_CURR_MODE),     PS := PGN_TO_PS(dwPGN1_CURR_MODE),     DST := ADR(abyCAN1RX_CURR_MODE),     RPT := T#0S, LIFE := , RESULT => , DEVICE => , LEN => );

  CAN1RX_COMMAND       (ENABLE := 1, CONFIG := bInit, PG := 0, PF := PGN_TO_PF(dwPGN1_COMMAND),       PS := PGN_TO_PS(dwPGN1_COMMAND),       DST := ADR(abyCAN1RX_COMMAND),       RPT := T#0S, LIFE := , RESULT => , DEVICE => , LEN => );

  CAN1RX_Set_GN2TempManual   (ENABLE := 1, CONFIG := bInit, PG := 0, PF := PGN_TO_PF(dwPGN1_Set_GN2TempManual),   PS := PGN_TO_PS(dwPGN1_Set_GN2TempManual),   DST := ADR(abyCAN1RX_Set_GN2TempManual),   RPT := T#0S, LIFE := , RESULT => , DEVICE => , LEN => );
  CAN1RX_Set_GN2OverPres     (ENABLE := 1, CONFIG := bInit, PG := 0, PF := PGN_TO_PF(dwPGN1_Set_GN2OverPres),     PS := PGN_TO_PS(dwPGN1_Set_GN2OverPres),     DST := ADR(abyCAN1RX_Set_GN2OverPres),     RPT := T#0S, LIFE := , RESULT => , DEVICE => , LEN => );
  CAN1RX_Set_BoostPresManual (ENABLE := 1, CONFIG := bInit, PG := 0, PF := PGN_TO_PF(dwPGN1_Set_BoostPresManual), PS := PGN_TO_PS(dwPGN1_Set_BoostPresManual), DST := ADR(abyCAN1RX_Set_BoostPresManual), RPT := T#0S, LIFE := , RESULT => , DEVICE => , LEN => );
  CAN1RX_Set_GN2Rate         (ENABLE := 1, CONFIG := bInit, PG := 0, PF := PGN_TO_PF(dwPGN1_Set_GN2Rate),         PS := PGN_TO_PS(dwPGN1_Set_GN2Rate),         DST := ADR(abyCAN1RX_Set_GN2Rate),         RPT := T#0S, LIFE := , RESULT => , DEVICE => , LEN => );
  CAN1RX_Set_LN2SaturTemp    (ENABLE := 1, CONFIG := bInit, PG := 0, PF := PGN_TO_PF(dwPGN1_Set_LN2SaturTemp),    PS := PGN_TO_PS(dwPGN1_Set_LN2SaturTemp),    DST := ADR(abyCAN1RX_Set_LN2SaturTemp),    RPT := T#0S, LIFE := , RESULT => , DEVICE => , LEN => );

(*-----------------------------------------------------------------------------------------------------------------------------------------------------------------------------------*)
(*Смена адреса установки*)

IF CAN1RX_UNIT_ADDR.RESULT = 1 THEN instFRAMWrite(Enable := 1, DST := iMemAdrCurrCANAddr, LEN := 1, SRC := ADR(abyCAN1RX_UNIT_ADDR[0])); END_IF;

(*-----------------------------------------------------------------------------------------------------------------------------------------------------------------------------------*)
(*Заполняем энергонезависимый массив параметров каналов*)

IF CAN1RX_CHANNEL_INDEX.RESULT = 1 THEN instMemCpy(DST := ADR(dwControlCAN1RX_CHANNEL_INDEX), SRC := ADR(abyCAN1RX_CHANNEL_INDEX), LEN := 4); bControlCAN1RX_CHANNEL_INDEX := 1; END_IF;

(*Проверяем, что номер страницы попадает в допустимый диапазон*)

IF dwControlCAN1RX_CHANNEL_INDEX >= 0 AND dwControlCAN1RX_CHANNEL_INDEX <= 63 AND bControlCAN1RX_CHANNEL_INDEX = 1
THEN
	instFRAMWrite(Enable := 1, DST := iMemAdrCHANNEL_INDEX, LEN := 4, SRC := ADR(dwControlCAN1RX_CHANNEL_INDEX));
	dwCHANNEL_INDEX := dwControlCAN1RX_CHANNEL_INDEX;
	dwControlCAN1RX_PARAM00 := aPage_Channel[dwCHANNEL_INDEX].PARAM_00;
	dwControlCAN1RX_PARAM09 := aPage_Channel[dwCHANNEL_INDEX].PARAM_09;
	bControlCAN1RX_CHANNEL_INDEX := 0;
ELSE
	bControlCAN1RX_CHANNEL_INDEX := 0;
END_IF;

(*Проверяем, что тип канала и номер канала измерения попадает в допустимый диапазон и потом записываем в массим каналов*)

IF CAN1RX_PARAM00.RESULT = 1 THEN instMemCpy(DST := ADR(dwControlCAN1RX_PARAM00), SRC := ADR(abyCAN1RX_PARAM00), LEN := 4); bControlCAN1RX_PARAM00 := 1; END_IF;
IF CAN1RX_PARAM09.RESULT = 1 THEN instMemCpy(DST := ADR(dwControlCAN1RX_PARAM09), SRC := ADR(abyCAN1RX_PARAM09), LEN := 4); bControlCAN1RX_PARAM09 := 1; END_IF;

IF
	(dwControlCAN1RX_CHANNEL_INDEX >= 0 AND dwControlCAN1RX_CHANNEL_INDEX <= 63 AND dwControlCAN1RX_PARAM00 = 0 AND dwControlCAN1RX_PARAM09 > 0 AND dwControlCAN1RX_PARAM09 <= 16) OR
	(dwControlCAN1RX_CHANNEL_INDEX >= 0 AND dwControlCAN1RX_CHANNEL_INDEX <= 63 AND dwControlCAN1RX_PARAM00 = 1 AND dwControlCAN1RX_PARAM09 > 0 AND dwControlCAN1RX_PARAM09 <=  8) OR
	(dwControlCAN1RX_CHANNEL_INDEX >= 0 AND dwControlCAN1RX_CHANNEL_INDEX <= 63 AND dwControlCAN1RX_PARAM00 = 2 AND dwControlCAN1RX_PARAM09 > 0 AND dwControlCAN1RX_PARAM09 <=  8) OR
	(dwControlCAN1RX_CHANNEL_INDEX >= 0 AND dwControlCAN1RX_CHANNEL_INDEX <= 63 AND dwControlCAN1RX_PARAM00 = 3 AND dwControlCAN1RX_PARAM09 > 0 AND dwControlCAN1RX_PARAM09 <=  8) OR
	(dwControlCAN1RX_CHANNEL_INDEX >= 0 AND dwControlCAN1RX_CHANNEL_INDEX <= 63 AND dwControlCAN1RX_PARAM00 = 4 AND dwControlCAN1RX_PARAM09 > 0 AND dwControlCAN1RX_PARAM09 <=  8) OR
	(dwControlCAN1RX_CHANNEL_INDEX >= 0 AND dwControlCAN1RX_CHANNEL_INDEX <= 63 AND dwControlCAN1RX_PARAM00 = 5 AND dwControlCAN1RX_PARAM09 > 0 AND dwControlCAN1RX_PARAM09 <=  8) OR
	(dwControlCAN1RX_CHANNEL_INDEX >= 0 AND dwControlCAN1RX_CHANNEL_INDEX <= 63 AND dwControlCAN1RX_PARAM00 = 6 AND dwControlCAN1RX_PARAM09 > 0 AND dwControlCAN1RX_PARAM09 <=  8)
THEN
	IF bControlCAN1RX_PARAM00 = 1    THEN instFRAMWrite(Enable := 1, DST := iMemAdrArrayParam00 + DWORD_TO_INT(dwCHANNEL_INDEX) * 4, LEN := 4, SRC := ADR(abyCAN1RX_PARAM00)); bControlCAN1RX_PARAM00 := 0; END_IF;
	IF CAN1RX_PARAM01.RESULT = 1     THEN instFRAMWrite(Enable := 1, DST := iMemAdrArrayParam01 + DWORD_TO_INT(dwCHANNEL_INDEX) * 4, LEN := 4, SRC := ADR(abyCAN1RX_PARAM01)); END_IF;
	IF CAN1RX_PARAM02.RESULT = 1     THEN instFRAMWrite(Enable := 1, DST := iMemAdrArrayParam02 + DWORD_TO_INT(dwCHANNEL_INDEX) * 4, LEN := 4, SRC := ADR(abyCAN1RX_PARAM02)); END_IF;
	IF CAN1RX_PARAM03.RESULT = 1     THEN instFRAMWrite(Enable := 1, DST := iMemAdrArrayParam03 + DWORD_TO_INT(dwCHANNEL_INDEX) * 4, LEN := 4, SRC := ADR(abyCAN1RX_PARAM03)); END_IF;
	IF CAN1RX_PARAM04.RESULT = 1     THEN instFRAMWrite(Enable := 1, DST := iMemAdrArrayParam04 + DWORD_TO_INT(dwCHANNEL_INDEX) * 4, LEN := 4, SRC := ADR(abyCAN1RX_PARAM04)); END_IF;
	IF CAN1RX_PARAM05.RESULT = 1     THEN instFRAMWrite(Enable := 1, DST := iMemAdrArrayParam05 + DWORD_TO_INT(dwCHANNEL_INDEX) * 4, LEN := 4, SRC := ADR(abyCAN1RX_PARAM05)); END_IF;
	IF CAN1RX_PARAM06.RESULT = 1     THEN instFRAMWrite(Enable := 1, DST := iMemAdrArrayParam06 + DWORD_TO_INT(dwCHANNEL_INDEX) * 4, LEN := 4, SRC := ADR(abyCAN1RX_PARAM06)); END_IF;
	IF CAN1RX_PARAM07.RESULT = 1     THEN instFRAMWrite(Enable := 1, DST := iMemAdrArrayParam07 + DWORD_TO_INT(dwCHANNEL_INDEX) * 4, LEN := 4, SRC := ADR(abyCAN1RX_PARAM07)); END_IF;
  (*IF CAN1RX_PARAM08.RESULT = 1     THEN instFRAMWrite(Enable := 1, DST := iMemAdrArrayParam08 + DWORD_TO_INT(dwCHANNEL_INDEX) * 4, LEN := 4, SRC := ADR(abyCAN1RX_PARAM08)); END_IF;*)
	IF bControlCAN1RX_PARAM09 = 1    THEN instFRAMWrite(Enable := 1, DST := iMemAdrArrayParam09 + DWORD_TO_INT(dwCHANNEL_INDEX) * 4, LEN := 4, SRC := ADR(abyCAN1RX_PARAM09)); bControlCAN1RX_PARAM09 := 0; END_IF;
	IF CAN1RX_PARAM10.RESULT = 1     THEN instFRAMWrite(Enable := 1, DST := iMemAdrArrayParam10 + DWORD_TO_INT(dwCHANNEL_INDEX) * 4, LEN := 4, SRC := ADR(abyCAN1RX_PARAM10)); END_IF;
END_IF;

(*-----------------------------------------------------------------------------------------------------------------------------------------------------------------------------------*)
(*Смена текущего режима работы*)

IF CAN1RX_CURR_MODE.RESULT = 1 THEN instFRAMWrite(Enable := 1, DST := iMemAdrCurrMode, LEN := 4, SRC := ADR(abyCAN1RX_CURR_MODE)); bCurrModeChange := 1; END_IF;

(*Извлечение номера команды, установка флага "Получена новая команда"*)
IF CAN1RX_COMMAND.RESULT = 1     THEN instMemCpy(DST := ADR(diCommand), SRC := ADR(abyCAN1RX_COMMAND), LEN := 4); bCommand := 1; END_IF;

IF CAN1RX_Set_GN2TempManual.RESULT = 1   THEN instFRAMWrite(Enable := 1, DST := iMemAdrSet_GN2TempManual,   LEN := 4, SRC := ADR(abyCAN1RX_Set_GN2TempManual));   bSet_HydHeatPresManual := 1; END_IF;
IF CAN1RX_Set_GN2OverPres.RESULT = 1     THEN instFRAMWrite(Enable := 1, DST := iMemAdrSet_GN2OverPres,     LEN := 4, SRC := ADR(abyCAN1RX_Set_GN2OverPres));     END_IF;
IF CAN1RX_Set_BoostPresManual.RESULT = 1 THEN instFRAMWrite(Enable := 1, DST := iMemAdrSet_BoostPresManual, LEN := 4, SRC := ADR(abyCAN1RX_Set_BoostPresManual)); bSet_BoostPresManual := 1; END_IF;
IF CAN1RX_Set_GN2Rate.RESULT = 1         THEN instFRAMWrite(Enable := 1, DST := iMemAdrSet_GN2Rate,         LEN := 4, SRC := ADR(abyCAN1RX_Set_GN2Rate));         bSet_TriplexRPMManual := 1; END_IF;
IF CAN1RX_Set_LN2SaturTemp.RESULT = 1    THEN instFRAMWrite(Enable := 1, DST := iMemAdrSet_LN2SaturTemp,    LEN := 4, SRC := ADR(abyCAN1RX_Set_LN2SaturTemp));    END_IF;

(*-----------------------------------------------------------------------------------------------------------------------------------------------------------------------------------*)
(**)

IF bInit = 1
THEN
	rSet_GN2OverPres := 3.5;
	instFRAMWrite(Enable := 1, DST := iMemAdrSet_GN2OverPres, LEN := 4, SRC := ADR(rSet_GN2OverPres));
END_IF;

(*-----------------------------------------------------------------------------------------------------------------------------------------------------------------------------------*)
(*Обработка команд*)

IF bCommand = 1 THEN
	CASE diCommand OF
		(*Номер команды*)
		  1: bDefaultSettings     := 1;         (*Установка флага "Команда 01"*)
		  2: bStop                := 1;         (*Установка флага "Команда 02"*)
			 bStart               := NOT bStop;
		  4: bHornDisable         := 0;         (*Установка флага "Команда 04"*)
		  5: bBlockDisable        := 1;         (*Установка флага "Команда 05"*)
		  6: bBlockDisable        := 0;         (*Установка флага "Команда 06"*)
(* 		  7: bCommand_07;                       (*Установка флага "Команда 07"*)
		  8: bCommand_08;                       (*Установка флага "Команда 08"*)*)
          9: bResetErrors         := 1;         (*Установка флага "Команда 09"*)
         10: bResetTotalAmountGN2 := 1;         (*Установка флага "Команда 10"*)
         11: bResetErrorsECU      := 1;         (*Установка флага "Команда 11"*)
			 bResetErrorsBuf      := 1;
			 bResetErrorsECU1     := 1;
			 bResetErrorsECU2     := 1;
         12: bPressSensorRST      := 1;         (*Установка флага "Команда 12"*)
(*       13: bCommand_13;                       (*Установка флага "Команда 13"*)*)
(*       14: bCommand_14;                       (*Установка флага "Команда 14"*)*)
(*       15: bCommand_15;                       (*Установка флага "Команда 15"*)*)
(*       16: bCommand_16;                       (*Установка флага "Команда 16"*)*)
(*       17: bCommand_17;                       (*Установка флага "Команда 17"*)*)
(*       18: bCommand_18;                       (*Установка флага "Команда 18"*)*)
(*       19: bCommand_19;                       (*Установка флага "Команда 19"*)*)
(*       20: bCommand_20;                       (*Установка флага "Команда 20"*)*)
(*       21: bCommand_21;                       (*Установка флага "Команда 21"*)*)
(*       22: bCommand_22;                       (*Установка флага "Команда 22"*)*)
(*       24: bCommand_23;                       (*Установка флага "Команда 23"*)*)
(*       25: bCommand_24;                       (*Установка флага "Команда 24"*)*)
(*       26: bCommand_25;                       (*Установка флага "Команда 25"*)*)
(*       27: bCommand_26;                       (*Установка флага "Команда 26"*)*)
(*       28: bCommand_27;                       (*Установка флага "Команда 27"*)*)
(*       29: bCommand_28;                       (*Установка флага "Команда 28"*)*)
(*       30: bCommand_29;                       (*Установка флага "Команда 29"*)*)
(*       31: bCommand_30;                       (*Установка флага "Команда 30"*)*)
(*       32: bCommand_31;                       (*Установка флага "Команда 31"*)*)
		ELSE;
	END_CASE;
END_IF;

(*-----------------------------------------------------------------------------------------------------------------------------------------------------------------------------------*)
(*Обработка ошибок CAN J1939*)

(*Обработка ошибок CAN J1939, если отсутствуют сообщения*)
IF FALSE OR FALSE
THEN
	bCAN1_J1939Errors := 1;
ELSE
	bCAN1_J1939Errors := 0;
END_IF;

(*Обработка ошибок CAN J1939, если предупреждение CAN1_WARNING от контроллера (возможно, обрыв линии)*)
IF CAN1_WARNING = 1
THEN
	bCAN1_J1939NotActive := 1;
ELSE
	bCAN1_J1939NotActive := 0;
END_IF;
END_PROGRAM

(* POU AUX_MODULES/PGN_TO_PF, ST *)
FUNCTION PGN_TO_PF : BYTE

VAR_INPUT
	PGN : DWORD;
END_VAR

VAR
END_VAR
PGN_TO_PF := DWORD_TO_BYTE(SHR(PGN, 8));
END_FUNCTION

(* POU AUX_MODULES/PGN_TO_PS, ST *)
FUNCTION PGN_TO_PS : BYTE

VAR_INPUT
	PGN : DWORD;
END_VAR

VAR
END_VAR
PGN_TO_PS := DWORD_TO_BYTE(PGN);
END_FUNCTION

(* POU CAN2_J1939/CAN2_J1939_Receive_processing, ST *)
PROGRAM CAN2_J1939_Receive_processing

VAR_INPUT
	bInit                : BOOL;
END_VAR

VAR
(*Electronic Engine Controller 1 - EEC1, Engine Speed*)
	byResult_EEC1        : BYTE;
	byDevice_EEC1        : BYTE;
	wLen_EEC1            : WORD;
	dwID_Parameter_EEC1  : DWORD := 16#0CF00400;
	byAvailable_EEC1     : BYTE;
	bOverFlow_EEC1       : BOOL;
	wError_EEC1			 : WORD;

(*Electronic Transmission Controller 1 - ETC1, Torque Converter Lockup Engaged*)
	byResult_ETC1        : BYTE;
	byDevice_ETC1        : BYTE;
	wLen_ETC1            : WORD;
	dwID_Parameter_ETC1  : DWORD := 16#CF00206;
	byAvailable_ETC1     : BYTE;
	bOverFlow_ETC1       : BOOL;
	wError_ETC1			 : WORD;

(*Electronic Transmission Controller 2 - ETC2, Transmission Selected Gear, Transmission Current Gear*)
	byResult_ETC2        : BYTE;
	byDevice_ETC2        : BYTE;
	wLen_ETC2            : WORD;
	dwID_Parameter_ETC2  : DWORD := 16#18F00503;
	byAvailable_ETC2     : BYTE;
	bOverFlow_ETC2       : BOOL;
	wError_ETC2			 : WORD;
END_VAR
(*-----------------------------------------------------------------------------------------------------------------------------------------------------------------------------------*)
(*Принимаем сообщения CAN J1939*)

CAN2RX_EEC1(ENABLE := 1, CONFIG := bInit, PG := 0, PF := byPDUFormat_EEC1, PS := byPDUSpecific_EEC1, DST := ADR(abyCAN2_Receive_EEC1), RPT := tRPT_EEC1, LIFE := 50, RESULT => , DEVICE => , LEN => );
CAN2RX_ETC1(ENABLE := 1, CONFIG := bInit, PG := 0, PF := byPDUFormat_ETC1, PS := byPDUSpecific_ETC1, DST := ADR(abyCAN2_Receive_ETC1), RPT := tRPT_ETC1, LIFE := 10, RESULT => , DEVICE => , LEN => );
CAN2RX_ETC2(ENABLE := 1, CONFIG := bInit, PG := 0, PF := byPDUFormat_ETC2, PS := byPDUSpecific_ETC2, DST := ADR(abyCAN2_Receive_ETC2), RPT := tRPT_ETC2, LIFE := 10, RESULT => , DEVICE => , LEN => );
CAN2RX_TC1 (ENABLE := 1, CONFIG := bInit, PG := 0, PF := byPDUFormat_TC1,  PS := byPDUSpecific_TC1,  DST := ADR(abyCAN2_Receive_TC1),  RPT := tRPT_TC1,  LIFE := 10, RESULT => , DEVICE => , LEN => );

(*-----------------------------------------------------------------------------------------------------------------------------------------------------------------------------------*)
(*Electronic Engine Controller 1 - EEC1, Engine Speed*)

IF CAN2RX_EEC1.RESULT = 1
THEN
	diCurrentEngineRPM := (SHL(BYTE_TO_WORD(abyCAN2_Receive_EEC1[5]),8) OR BYTE_TO_WORD(abyCAN2_Receive_EEC1[4])) / 8; (*Engine Speed*);  (*НЕЯВНОЕ REAL TO WORD !!!*)

	(*diCurrentEngineRPM := 1800; (*ТЕСТ!!!!!!!!!!!!!!!!!!!!!!!!!!!!!!!!!!!!!!!*)*)

END_IF;

IF CAN2RX_EEC1.RESULT = 3 (*Если пакетов CAN долго нет, то обнуляем соответствующий параметр*)
THEN
	diCurrentEngineRPM := 0;
END_IF;

(*-----------------------------------------------------------------------------------------------------------------------------------------------------------------------------------*)
(*Electronic Transmission Controller 1 - ETC1, Torque Converter Lockup Engaged*)

IF CAN2RX_ETC1.RESULT = 1
THEN
	byTorqueConverterLockupEngaged := abyCAN2_Receive_ETC1[1] AND 2#00001100; (*Torque Converter Lockup Engaged*)
END_IF;

IF CAN2RX_ETC1.RESULT = 3 (*Если пакетов CAN долго нет, то обнуляем соответствующий параметр*)
THEN
	byTorqueConverterLockupEngaged := 0;(*НО ЭТО ПО ВОПРОСОМ !!!!*)
END_IF;

(*-----------------------------------------------------------------------------------------------------------------------------------------------------------------------------------*)
(*Electronic Transmission Controller 2 - ETC2, Transmission Selected Gear, Transmission Current Gear*)

IF CAN2RX_ETC2.RESULT = 1
THEN
	diCurrentNumberGear := abyCAN2_Receive_ETC2[4] - 125; (*Current Gear*)
	(*iSelectedNumberGear := abyCAN2_Receive_ETC2[1] - 125; (*Selected Gear*)*)
END_IF;

IF CAN2RX_ETC2.RESULT = 3 (*Если пакетов CAN долго нет, то обнуляем соответствующий параметр*)
THEN
	diCurrentNumberGear := 0;
END_IF;

(*-----------------------------------------------------------------------------------------------------------------------------------------------------------------------------------*)
(*Обработка ошибок CAN J1939*)

(*Обработка ошибок CAN J1939, если отсутствуют сообщения от двигателя или АКПП*)
IF CAN2RX_EEC1.RESULT = 3 OR (CAN2RX_ETC1.RESULT = 3 AND CAN2RX_ETC2.RESULT = 3)
THEN
	bCAN2_J1939Errors := 1;
ELSE
	bCAN2_J1939Errors := 0;
END_IF;

(*Обработка ошибок CAN J1939, если предупреждение CAN2_WARNING от контроллера (возможно, обрыв линии)*)
IF CAN2_WARNING = 1
THEN
	bCAN2_J1939NotActive := 1;
ELSE
	bCAN2_J1939NotActive := 0;
END_IF;
END_PROGRAM

(* POU CAN2_J1939/CAN2_J1939_DM_processing, ST *)
PROGRAM CAN2_J1939_DM_processing

VAR_INPUT
	bInit                        : BOOL;
END_VAR

VAR
	adwErrors_SPN_DM1            : ARRAY [1..32] OF DWORD;
	adwErrors_SPN_DM2            : ARRAY [1..32] OF DWORD;

	adwErrors_FMI_DM1            : ARRAY [1..32] OF DWORD;
	adwErrors_FMI_DM2            : ARRAY [1..32] OF DWORD;

	adwErrors_OC_DM1             : ARRAY [1..32] OF DWORD;
	adwErrors_OC_DM2             : ARRAY [1..32] OF DWORD;

	adwErrors_SPN_CM_DM1         : ARRAY [1..32] OF DWORD;
	adwErrors_SPN_CM_DM2         : ARRAY [1..32] OF DWORD;

	byMalfunctionLampStatus_DM1  : BYTE;
	byRedStopLampStatus_DM1      : BYTE;
	byAmberWarningLampStatus_DM1 : BYTE;
	byProtectLampStatus_DM1      : BYTE;

	byMalfunctionLampStatus_DM2  : BYTE;
	byRedStopLampStatus_DM2      : BYTE;
	byAmberWarningLampStatus_DM2 : BYTE;
	byProtectLampStatus_DM2      : BYTE;

	instMemCpy                   : MEMCPY;
	i                            : INT;
	n1                           : INT := 1;
	n2                           : INT := 1;
	k1                           : INT := 1;
	k2                           : INT := 1;

	bStopTransmitDM1             : BOOL := 0;
	bStopTransmitDM2             : BOOL := 0;
END_VAR
(*-----------------------------------------------------------------------------------------------------------------------------------------------------------------------------------*)
(*Принимаем сообщения CAN J1939*)

CAN2RX_DM1 (ENABLE := 1, CONFIG := bInit, PG := 0, PF := byPDUFormat_DM1,  PS := byPDUSpecific_DM1,  DST := ADR(abyCAN2_Receive_DM1),  RPT := tRPT_DM1,  LIFE := 100, RESULT => , DEVICE => , LEN => );
CAN2RX_DM2 (ENABLE := 1, CONFIG := bInit, PG := 0, PF := byPDUFormat_DM2,  PS := byPDUSpecific_DM2,  DST := ADR(abyCAN2_Receive_DM2),  RPT := tRPT_DM2,  LIFE := 100, RESULT => , DEVICE => , LEN => );

(*-----------------------------------------------------------------------------------------------------------------------------------------------------------------------------------*)
(*Обработка DM1 и DM2*)

IF CAN2RX_DM1.RESULT = 1 AND CAN2RX_DM1.DEVICE = 0
THEN
	byMalfunctionLampStatus_DM1  := SHR((2#11000000 AND abyCAN2_Receive_DM1[1]), 6);
	byRedStopLampStatus_DM1      := SHR((2#00110000 AND abyCAN2_Receive_DM1[1]), 4);
	byAmberWarningLampStatus_DM1 := SHR((2#00001100 AND abyCAN2_Receive_DM1[1]), 2);
	byProtectLampStatus_DM1      :=     (2#00000011 AND abyCAN2_Receive_DM1[1]);

	FOR i := 1 TO 32
	DO
		adwErrors_SPN_FMI_DM1[i] := 0;
		adwErrors_SPN_DM1[i]     := 0;
		adwErrors_FMI_DM1[i]     := 0;
		adwErrors_OC_DM1[i]      := 0;
		adwErrors_SPN_CM_DM1[i]  := 0;
	END_FOR;

	(*byErrorsQty_DM1 := 0;*)

	byErrorsQty_DM1 := WORD_TO_BYTE(CAN2RX_DM1.LEN - 2) / 4;

	instMemCpy(DST := ADR(adwErrors_SPN_FMI_DM1[1]), SRC := ADR(abyCAN2_Receive_DM1[3]), LEN := (CAN2RX_DM1.LEN - 2));

	FOR i := 1 TO byErrorsQty_DM1
	DO
		adwErrors_SPN_DM1[i]    := SHR((2#0000000011100000_0000000000000000 AND adwErrors_SPN_FMI_DM1[i]),  5) OR (2#0000000000000000_1111111111111111 AND adwErrors_SPN_FMI_DM1[i]);
		adwErrors_FMI_DM1[i]    := SHR((2#0000000000011111_0000000000000000 AND adwErrors_SPN_FMI_DM1[i]), 16);
		adwErrors_OC_DM1[i]     := SHR((2#0111111100000000_0000000000000000 AND adwErrors_SPN_FMI_DM1[i]), 24);
		adwErrors_SPN_CM_DM1[i] := SHR((2#1000000000000000_0000000000000000 AND adwErrors_SPN_FMI_DM1[i]), 31);

		(*IF adwErrors_SPN_DM1[i] <> 0 THEN byErrorsQty_DM1 := byErrorsQty_DM1 + 1; END_IF;*)
	END_FOR;
END_IF;

IF CAN2RX_DM2.RESULT = 1 AND CAN2RX_DM2.DEVICE = 0
THEN
	byMalfunctionLampStatus_DM2  := SHR((2#11000000 AND abyCAN2_Receive_DM2[1]), 6);
	byRedStopLampStatus_DM2      := SHR((2#00110000 AND abyCAN2_Receive_DM2[1]), 4);
	byAmberWarningLampStatus_DM2 := SHR((2#00001100 AND abyCAN2_Receive_DM2[1]), 2);
	byProtectLampStatus_DM2      :=     (2#00000011 AND abyCAN2_Receive_DM2[1]);

	FOR i := 1 TO 32
	DO
		adwErrors_SPN_FMI_DM2[i] := 0;
		adwErrors_SPN_DM2[i]     := 0;
		adwErrors_FMI_DM2[i]     := 0;
		adwErrors_OC_DM2[i]      := 0;
		adwErrors_SPN_CM_DM2[i]  := 0;
	END_FOR;

	(*byErrorsQty_DM2 := 0;*)

	byErrorsQty_DM2 := WORD_TO_BYTE(CAN2RX_DM2.LEN - 2) / 4;

	instMemCpy(DST := ADR(adwErrors_SPN_FMI_DM2[1]), SRC := ADR(abyCAN2_Receive_DM2[3]), LEN := (CAN2RX_DM2.LEN - 2));

	FOR i := 1 TO byErrorsQty_DM2
	DO
		adwErrors_SPN_DM2[i]    := SHR((2#0000000011100000_0000000000000000 AND adwErrors_SPN_FMI_DM2[i]),  5) OR (2#0000000000000000_1111111111111111 AND adwErrors_SPN_FMI_DM2[i]);
		adwErrors_FMI_DM2[i]    := SHR((2#0000000000011111_0000000000000000 AND adwErrors_SPN_FMI_DM2[i]), 16);
		adwErrors_OC_DM2[i]     := SHR((2#0111111100000000_0000000000000000 AND adwErrors_SPN_FMI_DM2[i]), 24);
		adwErrors_SPN_CM_DM2[i] := SHR((2#1000000000000000_0000000000000000 AND adwErrors_SPN_FMI_DM2[i]), 31);

		(*IF adwErrors_SPN_DM2[i] <> 0 THEN byErrorsQty_DM2 := byErrorsQty_DM2 + 1; END_IF;*)
	END_FOR;
END_IF;

(*-----------------------------------------------------------------------------------------------------------------------------------------------------------------------------------*)
(**)

IF bResetErrorsBuf = 1
THEN

	FOR i := 1 TO 32
	DO
		(*adwErrors_SPN_FMI_DM2[i] := 0;*)
		adwErrors_SPN_DM2[i]     := 0;
		adwErrors_FMI_DM2[i]     := 0;
		adwErrors_OC_DM2[i]      := 0;
		adwErrors_SPN_CM_DM2[i]  := 0;
	END_FOR;

	FOR i := 1 TO 130
	DO
		abyCAN2_Receive_DM2[i] := 0;
	END_FOR;

	byErrorsQty_DM2 := 0;

	bResetErrorsBuf := 0;
END_IF;

(*-----------------------------------------------------------------------------------------------------------------------------------------------------------------------------------*)
(**)

byLampStateDM1 := 0;
byLampStateDM1 := byLampStateDM1 OR SHL(byMalfunctionLampStatus_DM1,  6);
byLampStateDM1 := byLampStateDM1 OR SHL(byRedStopLampStatus_DM1,      4);
byLampStateDM1 := byLampStateDM1 OR SHL(byAmberWarningLampStatus_DM1, 2);
byLampStateDM1 := byLampStateDM1 OR    (byProtectLampStatus_DM1        );

byLampStateDM2 := 0;
byLampStateDM2 := byLampStateDM2 OR SHL(byMalfunctionLampStatus_DM2,  6);
byLampStateDM2 := byLampStateDM2 OR SHL(byRedStopLampStatus_DM2,      4);
byLampStateDM2 := byLampStateDM2 OR SHL(byAmberWarningLampStatus_DM2, 2);
byLampStateDM2 := byLampStateDM2 OR    (byProtectLampStatus_DM2        );

instMemCpy(DST := ADR(abyCAN1TX_DM1_DESCR[0]), SRC := ADR(byErrorsQty_DM1), LEN := 1);
instMemCpy(DST := ADR(abyCAN1TX_DM2_DESCR[0]), SRC := ADR(byErrorsQty_DM2), LEN := 1);

instMemCpy(DST := ADR(abyCAN1TX_DM1_DESCR[1]), SRC := ADR(byLampStateDM1), LEN := 1);
instMemCpy(DST := ADR(abyCAN1TX_DM2_DESCR[1]), SRC := ADR(byLampStateDM2), LEN := 1);

IF CAN1TX_DM1_DESCR.RESULT = 1
THEN

	bStopTransmitDM1 := 0;

	FOR n1 := 1 TO 32 DO
		aCAN1ErrorDM1[n1].dwSPN       := adwErrors_SPN_DM1[n1];
		aCAN1ErrorDM1[n1].byFMI       := DWORD_TO_BYTE(adwErrors_FMI_DM1[n1]);
		aCAN1ErrorDM1[n1].byOC        := DWORD_TO_BYTE(adwErrors_OC_DM1[n1]);
		aCAN1ErrorDM1[n1].byErrorsQty := 0;
		aCAN1ErrorDM1[n1].byLampState := 0;
	END_FOR;
END_IF;

IF CAN1TX_DM2_DESCR.RESULT = 1
THEN

	bStopTransmitDM2 := 0;

	FOR n2 := 1 TO 32 DO
		aCAN1ErrorDM2[n2].dwSPN       := adwErrors_SPN_DM2[n2];
		aCAN1ErrorDM2[n2].byFMI       := DWORD_TO_BYTE(adwErrors_FMI_DM2[n2]);
		aCAN1ErrorDM2[n2].byOC        := DWORD_TO_BYTE(adwErrors_OC_DM2[n2]);
		aCAN1ErrorDM2[n2].byErrorsQty := 0;
		aCAN1ErrorDM2[n2].byLampState := 0;
	END_FOR;
END_IF;

(*-----------------------------------------------------------------------------------------------------------------------------------------------------------------------------------*)
(**)

IF byErrorsQty_DM1 = 0 OR bStopTransmitDM1 = 1 THEN bEnableTransmit_DM1 := 0; ELSE bEnableTransmit_DM1 := 1; END_IF;
IF byErrorsQty_DM2 = 0 OR bStopTransmitDM2 = 1 THEN bEnableTransmit_DM2 := 0; ELSE bEnableTransmit_DM2 := 1; END_IF;

instMemCpy(DST := ADR(abyDataCurrentDM1[1]), SRC := ADR(aCAN1ErrorDM1[k1]), LEN := 8);
IF CAN1TX_DM1.RESULT = 1 THEN k1 := k1 + 1; END_IF;
IF k1 > byErrorsQty_DM1 THEN k1 := 1; bStopTransmitDM1 := 1; END_IF;

instMemCpy(DST := ADR(abyDataCurrentDM2[1]), SRC := ADR(aCAN1ErrorDM2[k2]), LEN := 8);
IF CAN1TX_DM2.RESULT = 1 THEN k2 := k2 + 1; END_IF;
IF k2 > byErrorsQty_DM2 THEN k2 := 1; bStopTransmitDM2 := 1; END_IF;
END_PROGRAM

(* POU CAN1_J1939/CAN1_J1939_Output_processing, ST *)
 PROGRAM CAN1_J1939_Output_processing

VAR_INPUT
	bInit      : BOOL;
END_VAR

VAR
	instMemCpy : MEMCPY;
END_VAR
(*-----------------------------------------------------------------------------------------------------------------------------------------------------------------------------------*)
(**)

instMemCpy(DST := ADR(abyCAN1TX_UNIT_ADDR     [0]), SRC := ADR(byCurrCAN1Addr),                          LEN := 1);(*Адрес установки*)

instMemCpy(DST := ADR(abyCAN1TX_CHANNEL_INDEX [0]), SRC := ADR(dwCHANNEL_INDEX),                         LEN := 4);(*Номер текущего канала*)
instMemCpy(DST := ADR(abyCAN1TX_PARAM00       [0]), SRC := ADR(aPage_Channel[dwCHANNEL_INDEX].PARAM_00), LEN := 4);(**)
instMemCpy(DST := ADR(abyCAN1TX_PARAM01       [0]), SRC := ADR(aPage_Channel[dwCHANNEL_INDEX].PARAM_01), LEN := 4);(**)
instMemCpy(DST := ADR(abyCAN1TX_PARAM02       [0]), SRC := ADR(aPage_Channel[dwCHANNEL_INDEX].PARAM_02), LEN := 4);(**)
instMemCpy(DST := ADR(abyCAN1TX_PARAM03       [0]), SRC := ADR(aPage_Channel[dwCHANNEL_INDEX].PARAM_03), LEN := 4);(**)
instMemCpy(DST := ADR(abyCAN1TX_PARAM04       [0]), SRC := ADR(aPage_Channel[dwCHANNEL_INDEX].PARAM_04), LEN := 4);(*Времена усреднения каналов*)
instMemCpy(DST := ADR(abyCAN1TX_PARAM05       [0]), SRC := ADR(aPage_Channel[dwCHANNEL_INDEX].PARAM_05), LEN := 4);(*Коэффициенты, учитывающие особенности механики*)
instMemCpy(DST := ADR(abyCAN1TX_PARAM06       [0]), SRC := ADR(aPage_Channel[dwCHANNEL_INDEX].PARAM_06), LEN := 4);(*Описания каналов*)
instMemCpy(DST := ADR(abyCAN1TX_PARAM07       [0]), SRC := ADR(aPage_Channel[dwCHANNEL_INDEX].PARAM_07), LEN := 4);(**)
instMemCpy(DST := ADR(abyCAN1TX_PARAM08       [0]), SRC := ADR(aPage_Channel[dwCHANNEL_INDEX].PARAM_08), LEN := 4);(*Необработанное значения канала*)
instMemCpy(DST := ADR(abyCAN1TX_PARAM09       [0]), SRC := ADR(aPage_Channel[dwCHANNEL_INDEX].PARAM_09), LEN := 4);(**)
instMemCpy(DST := ADR(abyCAN1TX_PARAM10       [0]), SRC := ADR(aPage_Channel[dwCHANNEL_INDEX].PARAM_10), LEN := 4);(**)

instMemCpy(DST := ADR(abyCAN1TX_CURR_MODE         [0]), SRC := ADR(dwCurrMode),                          LEN := 4);(**)

instMemCpy(DST:=ADR(abyCAN1TX_TOTAL_TIME          [0]), SRC:=ADR(rTotalServiceMeterOut),                 LEN:=4);(*Счетчик моточасов, суммарно за все время работы*)
instMemCpy(DST:=ADR(abyCAN1TX_LAST_TIME           [0]), SRC:=ADR(rLastServiceMeterOut),                  LEN:=4);(*Счетчик моточасов, с момента последнего включения*)

instMemCpy(DST:=ADR(abyCAN1TX_COMMAND             [0]), SRC:=ADR(diCommand),                             LEN:=4);(**)

instMemCpy(DST:=ADR(abyCAN1TX_STATE_ADC_MS        [0]), SRC:=ADR(dwErrorADC_MS),                         LEN:=4);(*Обрывы и короткие замыкания по входам аналоговых каналов*)
instMemCpy(DST:=ADR(abyCAN1TX_STATE_ADC_SL1       [0]), SRC:=ADR(dwErrorADC_SL1),                        LEN:=4);(*Обрывы и короткие замыкания по входам аналоговых каналов*)
instMemCpy(DST:=ADR(abyCAN1TX_STATE_ADC_SL2       [0]), SRC:=ADR(dwErrorADC_SL2),                        LEN:=4);(*Обрывы и короткие замыкания по входам аналоговых каналов*)
instMemCpy(DST:=ADR(abyCAN1TX_STATE_ADC_SL3       [0]), SRC:=ADR(dwErrorADC_SL3),                        LEN:=4);(*Обрывы и короткие замыкания по входам аналоговых каналов*)

instMemCpy(DST:=ADR(abyCAN1TX_MS_SV               [0]), SRC:=ADR(rECU_SupplyVoltage),                    LEN:=4);(*Напряжение питания контроллера Master*)
instMemCpy(DST:=ADR(abyCAN1TX_MS_T                [0]), SRC:=ADR(rECU_Temperature),                      LEN:=4);(*Tемпература контроллера Master*)
instMemCpy(DST:=ADR(abyCAN1TX_PROG_CRC_MS         [0]), SRC:=ADR(dwMS_ProgramCRC),                       LEN:=4);(*Идентификатор CRC программы контроллера Master*)
instMemCpy(DST:=ADR(abyCAN1TX_PROG_ID_MS          [0]), SRC:=ADR(abyMS_ProgramID),                       LEN:=4);(*Идентификатор программы контроллера Master*)

instMemCpy(DST:=ADR(abyCAN1TX_STATE_MS            [0]), SRC:=ADR(abyDataStateMS),                        LEN:=4);(*Ошибки контроллера Master*)
instMemCpy(DST:=ADR(abyCAN1TX_STATE_SL1           [0]), SRC:=ADR(abyDataStateSL1),                       LEN:=4);(*Ошибки контроллера Slave 1*)
instMemCpy(DST:=ADR(abyCAN1TX_STATE_SL2           [0]), SRC:=ADR(abyDataStateSL2),                       LEN:=4);(*Ошибки контроллера Slave 2*)
instMemCpy(DST:=ADR(abyCAN1TX_STATE_SL3           [0]), SRC:=ADR(abyDataStateSL3),                       LEN:=4);(*Ошибки контроллера Slave 3*)

instMemCpy(DST:=ADR(abyCAN1TX_DM1                 [0]), SRC:=ADR(abyDataCurrentDM1),                     LEN:=8);(**)
instMemCpy(DST:=ADR(abyCAN1TX_DM2                 [0]), SRC:=ADR(abyDataCurrentDM2),                     LEN:=8);(**)

rWF_PresOut := rIW_GN2_Pres - rWF_PresCor;

instMemCpy(DST:=ADR(abyCAN1TX_GN2_Temp            [0]), SRC:=ADR(rIW_GN2_Temp),                          LEN:=4);(*Температура нагнетания*)
instMemCpy(DST:=ADR(abyCAN1TX_WF_PresOut          [0]), SRC:=ADR(rWF_PresOut),                           LEN:=4);(*Давление нагнетания*)
instMemCpy(DST:=ADR(abyCAN1TX_LN2_Temp            [0]), SRC:=ADR(rIW_LN2_Temp),                          LEN:=4);(*Температура азота жидкого*)
instMemCpy(DST:=ADR(abyCAN1TX_BoostPres           [0]), SRC:=ADR(rIW_BoostPres),                         LEN:=4);(*Давление подпитки*)
instMemCpy(DST:=ADR(abyCAN1TX_HydHeatPres         [0]), SRC:=ADR(rIW_HydHeatPres),                       LEN:=4);(*Давление гидронагрева*)
instMemCpy(DST:=ADR(abyCAN1TX_CoolTempIn          [0]), SRC:=ADR(rIW_CoolTempIn),                        LEN:=4);(*Температура ОЖ до испарителя*)
instMemCpy(DST:=ADR(abyCAN1TX_CoolTempInMin       [0]), SRC:=ADR(rCoolTempInMin),                        LEN:=4);(*Температура предварительного прогрева ОЖ*)

instMemCpy(DST:=ADR(abyCAN1TX_TriplexRPM          [0]), SRC:=ADR(rFRQ_TriplexRPM),                       LEN:=4);(*Обороты НВД*)

instMemCpy(DST:=ADR(abyCAN1TX_InputState          [0]), SRC:=ADR(dwInputState),                          LEN:=4);(*Дискретные входы*)
instMemCpy(DST:=ADR(abyCAN1TX_OutputState         [0]), SRC:=ADR(dwOutputState),                         LEN:=4);(*Дискретные выходы*)
instMemCpy(DST:=ADR(abyCAN1TX_Current_GN2Rate     [0]), SRC:=ADR(rCurrent_GN2Rate),                      LEN:=4);(*Производительность установки*)
instMemCpy(DST:=ADR(abyCAN1TX_TotalAmountGN2      [0]), SRC:=ADR(rTotalAmountGN2),                       LEN:=4);(*Общий объем закачанного азота*)
instMemCpy(DST:=ADR(abyCAN1TX_CurrEngineRPM       [0]), SRC:=ADR(diCurrentEngineRPM),                    LEN:=4);(*Обороты двигателя*)
instMemCpy(DST:=ADR(abyCAN1TX_CurrNumberGear      [0]), SRC:=ADR(diCurrentNumberGear),                   LEN:=4);(*Номер передачи АКПП*)

instMemCpy(DST:=ADR(abyCAN1TX_Set_GN2TempManual   [0]), SRC:=ADR(rSet_GN2TempManual),                    LEN:=4);(*Установочные значения. Температура азота*)
instMemCpy(DST:=ADR(abyCAN1TX_Set_GN2OverPres     [0]), SRC:=ADR(rSet_GN2OverPres),                      LEN:=4);(*Установочные значения. Предельно допустимое давление азота на выходе*)
instMemCpy(DST:=ADR(abyCAN1TX_Set_BoostPresManual [0]), SRC:=ADR(rSet_BoostPresManual),                  LEN:=4);(*Установочные значения. Давление подпитки в ручном режиме*)
instMemCpy(DST:=ADR(abyCAN1TX_Set_GN2Rate         [0]), SRC:=ADR(rSet_GN2Rate),                          LEN:=4);(*Установочные значения. Производительность установки*)
instMemCpy(DST:=ADR(abyCAN1TX_Set_LN2SaturTemp    [0]), SRC:=ADR(rSet_LN2SaturTemp),                     LEN:=4);(*Установочные значения. Температура азота, когда можно переходить к управлению подкачивающим насосом*)
instMemCpy(DST:=ADR(abyCAN1TX_ReqStageOper        [0]), SRC:=ADR(diRequiredStageOperation),              LEN:=4);(*Требуемый этап работы*)
instMemCpy(DST:=ADR(abyCAN1TX_CurStageOper        [0]), SRC:=ADR(wCurrentStageOperation),                LEN:=4);(*Текущий этап работы*)

instMemCpy(DST:=ADR(abyCAN1TX_ErrorState          [0]), SRC:=ADR(dwErrorState),                          LEN:=4);(*Сообщения*)
instMemCpy(DST:=ADR(abyCAN1TX_ProcessState        [0]), SRC:=ADR(dwProcessState),                        LEN:=4);(*Состояние процесса*)

instMemCpy(DST:=ADR(abyCAN1TX_GN2_Pres            [0]), SRC:=ADR(rIW_GN2_Pres),                          LEN:=4);(**)
END_PROGRAM

(* POU CAN1_J1939/CAN1_J1939_Transmit_processing, ST *)
PROGRAM CAN1_J1939_Transmit_processing

VAR_INPUT
	bInit : BOOL;
END_VAR

VAR
END_VAR
(*-----------------------------------------------------------------------------------------------------------------------------------------------------------------------------------*)
(**)

CAN1TX_UNIT_ADDR     (ENABLE := 1, Prio := 6, PG := 0, PF := PGN_TO_PF(dwPGN1_UNIT_ADDR),     PS := PGN_TO_PS(dwPGN1_UNIT_ADDR),     SRC := ADR(abyCAN1TX_UNIT_ADDR),     LEN := 8, RPT := T#1S, RESULT => );

CAN1TX_CHANNEL_INDEX (ENABLE := 1, Prio := 6, PG := 0, PF := PGN_TO_PF(dwPGN1_CHANNEL_INDEX), PS := PGN_TO_PS(dwPGN1_CHANNEL_INDEX), SRC := ADR(abyCAN1TX_CHANNEL_INDEX), LEN := 8, RPT := T#1S, RESULT => );
CAN1TX_PARAM00       (ENABLE := 1, Prio := 6, PG := 0, PF := PGN_TO_PF(dwPGN1_PARAM00),       PS := PGN_TO_PS(dwPGN1_PARAM00),       SRC := ADR(abyCAN1TX_PARAM00),       LEN := 8, RPT := T#1S, RESULT => );
CAN1TX_PARAM01       (ENABLE := 1, Prio := 6, PG := 0, PF := PGN_TO_PF(dwPGN1_PARAM01),       PS := PGN_TO_PS(dwPGN1_PARAM01),       SRC := ADR(abyCAN1TX_PARAM01),       LEN := 8, RPT := T#1S, RESULT => );
CAN1TX_PARAM02       (ENABLE := 1, Prio := 6, PG := 0, PF := PGN_TO_PF(dwPGN1_PARAM02),       PS := PGN_TO_PS(dwPGN1_PARAM02),       SRC := ADR(abyCAN1TX_PARAM02),       LEN := 8, RPT := T#1S, RESULT => );
CAN1TX_PARAM03       (ENABLE := 1, Prio := 6, PG := 0, PF := PGN_TO_PF(dwPGN1_PARAM03),       PS := PGN_TO_PS(dwPGN1_PARAM03),       SRC := ADR(abyCAN1TX_PARAM03),       LEN := 8, RPT := T#1S, RESULT => );
CAN1TX_PARAM04       (ENABLE := 1, Prio := 6, PG := 0, PF := PGN_TO_PF(dwPGN1_PARAM04),       PS := PGN_TO_PS(dwPGN1_PARAM04),       SRC := ADR(abyCAN1TX_PARAM04),       LEN := 8, RPT := T#1S, RESULT => );
CAN1TX_PARAM05       (ENABLE := 1, Prio := 6, PG := 0, PF := PGN_TO_PF(dwPGN1_PARAM05),       PS := PGN_TO_PS(dwPGN1_PARAM05),       SRC := ADR(abyCAN1TX_PARAM05),       LEN := 8, RPT := T#1S, RESULT => );
CAN1TX_PARAM06       (ENABLE := 1, Prio := 6, PG := 0, PF := PGN_TO_PF(dwPGN1_PARAM06),       PS := PGN_TO_PS(dwPGN1_PARAM06),       SRC := ADR(abyCAN1TX_PARAM06),       LEN := 8, RPT := T#1S, RESULT => );
CAN1TX_PARAM07       (ENABLE := 1, Prio := 6, PG := 0, PF := PGN_TO_PF(dwPGN1_PARAM07),       PS := PGN_TO_PS(dwPGN1_PARAM07),       SRC := ADR(abyCAN1TX_PARAM07),       LEN := 8, RPT := T#1S, RESULT => );
CAN1TX_PARAM08       (ENABLE := 1, Prio := 6, PG := 0, PF := PGN_TO_PF(dwPGN1_PARAM08),       PS := PGN_TO_PS(dwPGN1_PARAM08),       SRC := ADR(abyCAN1TX_PARAM08),       LEN := 8, RPT := T#1S, RESULT => );
CAN1TX_PARAM09       (ENABLE := 1, Prio := 6, PG := 0, PF := PGN_TO_PF(dwPGN1_PARAM09),       PS := PGN_TO_PS(dwPGN1_PARAM09),       SRC := ADR(abyCAN1TX_PARAM09),       LEN := 8, RPT := T#1S, RESULT => );
CAN1TX_PARAM10       (ENABLE := 1, Prio := 6, PG := 0, PF := PGN_TO_PF(dwPGN1_PARAM10),       PS := PGN_TO_PS(dwPGN1_PARAM10),       SRC := ADR(abyCAN1TX_PARAM10),       LEN := 8, RPT := T#1S, RESULT => );

CAN1TX_CURR_MODE     (ENABLE := 1, Prio := 6, PG := 0, PF := PGN_TO_PF(dwPGN1_CURR_MODE),     PS := PGN_TO_PS(dwPGN1_CURR_MODE),     SRC := ADR(abyCAN1TX_CURR_MODE),     LEN := 8, RPT := T#1S, RESULT => );

CAN1TX_TOTAL_TIME     (ENABLE := 1, Prio := 6, PG := 0, PF := PGN_TO_PF(dwPGN1_TOTAL_TIME),      PS := PGN_TO_PS(dwPGN1_TOTAL_TIME),      SRC := ADR(abyCAN1TX_TOTAL_TIME),      LEN := 8, RPT := T#1S,   RESULT => );
CAN1TX_LAST_TIME      (ENABLE := 1, Prio := 6, PG := 0, PF := PGN_TO_PF(dwPGN1_LAST_TIME),       PS := PGN_TO_PS(dwPGN1_LAST_TIME),       SRC := ADR(abyCAN1TX_LAST_TIME),       LEN := 8, RPT := T#1S,   RESULT => );

CAN1TX_COMMAND        (ENABLE := 1, Prio := 6, PG := 0, PF := PGN_TO_PF(dwPGN1_COMMAND),         PS := PGN_TO_PS(dwPGN1_COMMAND),         SRC := ADR(abyCAN1TX_COMMAND),         LEN := 8, RPT := T#0.5S, RESULT => );

CAN1TX_STATE_ADC_MS   (ENABLE := 1, Prio := 6, PG := 0, PF := PGN_TO_PF(dwPGN1_STATE_ADC_MS),    PS := PGN_TO_PS(dwPGN1_STATE_ADC_MS),    SRC := ADR(abyCAN1TX_STATE_ADC_MS),    LEN := 8, RPT := T#1S,   RESULT => );
CAN1TX_STATE_ADC_SL1  (ENABLE := 1, Prio := 6, PG := 0, PF := PGN_TO_PF(dwPGN1_STATE_ADC_SL1),   PS := PGN_TO_PS(dwPGN1_STATE_ADC_SL1),   SRC := ADR(abyCAN1TX_STATE_ADC_SL1),   LEN := 8, RPT := T#1S,   RESULT => );
CAN1TX_STATE_ADC_SL2  (ENABLE := 1, Prio := 6, PG := 0, PF := PGN_TO_PF(dwPGN1_STATE_ADC_SL2),   PS := PGN_TO_PS(dwPGN1_STATE_ADC_SL2),   SRC := ADR(abyCAN1TX_STATE_ADC_SL2),   LEN := 8, RPT := T#1S,   RESULT => );
CAN1TX_STATE_ADC_SL3  (ENABLE := 1, Prio := 6, PG := 0, PF := PGN_TO_PF(dwPGN1_STATE_ADC_SL3),   PS := PGN_TO_PS(dwPGN1_STATE_ADC_SL3),   SRC := ADR(abyCAN1TX_STATE_ADC_SL3),   LEN := 8, RPT := T#1S,   RESULT => );

CAN1TX_MS_SV          (ENABLE := 1, Prio := 6, PG := 0, PF := PGN_TO_PF(dwPGN1_MS_SV),           PS := PGN_TO_PS(dwPGN1_MS_SV),           SRC := ADR(abyCAN1TX_MS_SV),           LEN := 8, RPT := T#1S,   RESULT => );
CAN1TX_MS_T           (ENABLE := 1, Prio := 6, PG := 0, PF := PGN_TO_PF(dwPGN1_MS_T),            PS := PGN_TO_PS(dwPGN1_MS_T),            SRC := ADR(abyCAN1TX_MS_T),            LEN := 8, RPT := T#1S,   RESULT => );
CAN1TX_PROG_CRC_MS    (ENABLE := 1, Prio := 6, PG := 0, PF := PGN_TO_PF(dwPGN1_PROG_CRC_MS),     PS := PGN_TO_PS(dwPGN1_PROG_CRC_MS),     SRC := ADR(abyCAN1TX_PROG_CRC_MS),     LEN := 8, RPT := T#1S,   RESULT => );
CAN1TX_PROG_ID_MS     (ENABLE := 1, Prio := 6, PG := 0, PF := PGN_TO_PF(dwPGN1_PROG_ID_MS),      PS := PGN_TO_PS(dwPGN1_PROG_ID_MS),      SRC := ADR(abyCAN1TX_PROG_ID_MS),      LEN := 8, RPT := T#1S,   RESULT => );

CAN1TX_STATE_MS       (ENABLE := 1, Prio := 6, PG := 0, PF := PGN_TO_PF(dwPGN1_STATE_MS),        PS := PGN_TO_PS(dwPGN1_STATE_MS),        SRC := ADR(abyCAN1TX_STATE_MS),        LEN := 8, RPT := T#0.5S, RESULT => );
CAN1TX_STATE_SL1      (ENABLE := 1, Prio := 6, PG := 0, PF := PGN_TO_PF(dwPGN1_STATE_SL1),       PS := PGN_TO_PS(dwPGN1_STATE_SL1),       SRC := ADR(abyCAN1TX_STATE_SL1),       LEN := 8, RPT := T#0.5S, RESULT => );
CAN1TX_STATE_SL2      (ENABLE := 1, Prio := 6, PG := 0, PF := PGN_TO_PF(dwPGN1_STATE_SL2),       PS := PGN_TO_PS(dwPGN1_STATE_SL2),       SRC := ADR(abyCAN1TX_STATE_SL2),       LEN := 8, RPT := T#0.5S, RESULT => );
CAN1TX_STATE_SL3      (ENABLE := 1, Prio := 6, PG := 0, PF := PGN_TO_PF(dwPGN1_STATE_SL3),       PS := PGN_TO_PS(dwPGN1_STATE_SL3),       SRC := ADR(abyCAN1TX_STATE_SL3),       LEN := 8, RPT := T#0.5S, RESULT => );

CAN1TX_DM1            (ENABLE := bEnableTransmit_DM1, Prio := 6, PG := 0, PF := PGN_TO_PF(dwPGN1_DM1),       PS := PGN_TO_PS(dwPGN1_DM1),       SRC := ADR(abyCAN1TX_DM1),       LEN := 8, RPT := T#0.1S, RESULT => );
(*CAN1TX_DM2            (ENABLE := bEnableTransmit_DM2, Prio := 6, PG := 0, PF := PGN_TO_PF(dwPGN1_DM2),       PS := PGN_TO_PS(dwPGN1_DM2),       SRC := ADR(abyCAN1TX_DM2),       LEN := 8, RPT := T#0.1S, RESULT => );*)
CAN1TX_DM1_DESCR      (ENABLE := 1,                   Prio := 6, PG := 0, PF := PGN_TO_PF(dwPGN1_DM1_DESCR), PS := PGN_TO_PS(dwPGN1_DM1_DESCR), SRC := ADR(abyCAN1TX_DM1_DESCR), LEN := 8, RPT := T#5S,   RESULT => );
(*CAN1TX_DM2_DESCR      (ENABLE := 1,                   Prio := 6, PG := 0, PF := PGN_TO_PF(dwPGN1_DM2_DESCR), PS := PGN_TO_PS(dwPGN1_DM2_DESCR), SRC := ADR(abyCAN1TX_DM2_DESCR), LEN := 8, RPT := T#5S,   RESULT => );*)

CAN1TX_GN2_Temp       (ENABLE := 1, Prio := 6, PG := 0, PF := PGN_TO_PF(dwPGN1_GN2_Temp),                 PS := PGN_TO_PS(dwPGN1_GN2_Temp),            SRC := ADR(abyCAN1TX_GN2_Temp),            LEN := 8, RPT := T#0.5S, RESULT => );
CAN1TX_WF_PresOut     (ENABLE := 1, Prio := 6, PG := 0, PF := PGN_TO_PF(dwPGN1_WF_PresOut),               PS := PGN_TO_PS(dwPGN1_WF_PresOut),          SRC := ADR(abyCAN1TX_WF_PresOut),          LEN := 8, RPT := T#0.5S, RESULT => );
CAN1TX_LN2_Temp       (ENABLE := 1, Prio := 6, PG := 0, PF := PGN_TO_PF(dwPGN1_LN2_Temp),                 PS := PGN_TO_PS(dwPGN1_LN2_Temp),            SRC := ADR(abyCAN1TX_LN2_Temp),            LEN := 8, RPT := T#0.5S, RESULT => );
CAN1TX_BoostPres      (ENABLE := 1, Prio := 6, PG := 0, PF := PGN_TO_PF(dwPGN1_BoostPres),                PS := PGN_TO_PS(dwPGN1_BoostPres),           SRC := ADR(abyCAN1TX_BoostPres),           LEN := 8, RPT := T#0.5S, RESULT => );
CAN1TX_HydHeatPres    (ENABLE := 1, Prio := 6, PG := 0, PF := PGN_TO_PF(dwPGN1_HydHeatPres),              PS := PGN_TO_PS(dwPGN1_HydHeatPres),         SRC := ADR(abyCAN1TX_HydHeatPres),         LEN := 8, RPT := T#0.5S, RESULT => );
CAN1TX_CoolTempIn     (ENABLE := 1, Prio := 6, PG := 0, PF := PGN_TO_PF(dwPGN1_CoolTempIn),               PS := PGN_TO_PS(dwPGN1_CoolTempIn),          SRC := ADR(abyCAN1TX_CoolTempIn),          LEN := 8, RPT := T#0.5S, RESULT => );

CAN1TX_TriplexRPM     (ENABLE := 1, Prio := 6, PG := 0, PF := PGN_TO_PF(dwPGN1_TriplexRPM),               PS := PGN_TO_PS(dwPGN1_TriplexRPM),          SRC := ADR(abyCAN1TX_TriplexRPM),          LEN := 8, RPT := T#0.5S, RESULT => );

CAN1TX_InputState          (ENABLE := 1, Prio := 6, PG := 0, PF := PGN_TO_PF(dwPGN1_InputState),          PS := PGN_TO_PS(dwPGN1_InputState),          SRC := ADR(abyCAN1TX_InputState),          LEN := 8, RPT := T#0.5S,  RESULT => );
CAN1TX_OutputState         (ENABLE := 1, Prio := 6, PG := 0, PF := PGN_TO_PF(dwPGN1_OutputState),         PS := PGN_TO_PS(dwPGN1_OutputState),         SRC := ADR(abyCAN1TX_OutputState),         LEN := 8, RPT := T#0.05S, RESULT => );

CAN1TX_Current_GN2Rate     (ENABLE := 1, Prio := 6, PG := 0, PF := PGN_TO_PF(dwPGN1_Current_GN2Rate),     PS := PGN_TO_PS(dwPGN1_Current_GN2Rate),     SRC := ADR(abyCAN1TX_Current_GN2Rate),     LEN := 8, RPT := T#1S,    RESULT => );
CAN1TX_TotalAmountGN2      (ENABLE := 1, Prio := 6, PG := 0, PF := PGN_TO_PF(dwPGN1_TotalAmountGN2),      PS := PGN_TO_PS(dwPGN1_TotalAmountGN2),      SRC := ADR(abyCAN1TX_TotalAmountGN2),      LEN := 8, RPT := T#1S,    RESULT => );
CAN1TX_CurrEngineRPM       (ENABLE := 1, Prio := 6, PG := 0, PF := PGN_TO_PF(dwPGN1_CurrEngineRPM),       PS := PGN_TO_PS(dwPGN1_CurrEngineRPM),       SRC := ADR(abyCAN1TX_CurrEngineRPM),       LEN := 8, RPT := T#1S,    RESULT => );
CAN1TX_CurrNumberGear      (ENABLE := 1, Prio := 6, PG := 0, PF := PGN_TO_PF(dwPGN1_CurrNumberGear),      PS := PGN_TO_PS(dwPGN1_CurrNumberGear),      SRC := ADR(abyCAN1TX_CurrNumberGear),      LEN := 8, RPT := T#1S,    RESULT => );
CAN1TX_Set_GN2TempManual   (ENABLE := 1, Prio := 6, PG := 0, PF := PGN_TO_PF(dwPGN1_Set_GN2TempManual),   PS := PGN_TO_PS(dwPGN1_Set_GN2TempManual),   SRC := ADR(abyCAN1TX_Set_GN2TempManual),   LEN := 8, RPT := T#0.25S, RESULT => );
CAN1TX_Set_GN2OverPres     (ENABLE := 1, Prio := 6, PG := 0, PF := PGN_TO_PF(dwPGN1_Set_GN2OverPres),     PS := PGN_TO_PS(dwPGN1_Set_GN2OverPres),     SRC := ADR(abyCAN1TX_Set_GN2OverPres),     LEN := 8, RPT := T#0.25S, RESULT => );
CAN1TX_Set_BoostPresManual (ENABLE := 1, Prio := 6, PG := 0, PF := PGN_TO_PF(dwPGN1_Set_BoostPresManual), PS := PGN_TO_PS(dwPGN1_Set_BoostPresManual), SRC := ADR(abyCAN1TX_Set_BoostPresManual), LEN := 8, RPT := T#0.25S, RESULT => );
CAN1TX_Set_GN2Rate         (ENABLE := 1, Prio := 6, PG := 0, PF := PGN_TO_PF(dwPGN1_Set_GN2Rate),         PS := PGN_TO_PS(dwPGN1_Set_GN2Rate),         SRC := ADR(abyCAN1TX_Set_GN2Rate),         LEN := 8, RPT := T#0.25S, RESULT => );
CAN1TX_Set_LN2SaturTemp    (ENABLE := 1, Prio := 6, PG := 0, PF := PGN_TO_PF(dwPGN1_Set_LN2SaturTemp),    PS := PGN_TO_PS(dwPGN1_Set_LN2SaturTemp),    SRC := ADR(abyCAN1TX_Set_LN2SaturTemp),    LEN := 8, RPT := T#0.25S, RESULT => );
CAN1TX_ReqStageOper        (ENABLE := 1, Prio := 6, PG := 0, PF := PGN_TO_PF(dwPGN1_ReqStageOper),        PS := PGN_TO_PS(dwPGN1_ReqStageOper),        SRC := ADR(abyCAN1TX_ReqStageOper),        LEN := 8, RPT := T#1S,    RESULT => );
CAN1TX_CurStageOper        (ENABLE := 1, Prio := 6, PG := 0, PF := PGN_TO_PF(dwPGN1_CurStageOper),        PS := PGN_TO_PS(dwPGN1_CurStageOper),        SRC := ADR(abyCAN1TX_CurStageOper),        LEN := 8, RPT := T#1S,    RESULT => );
CAN1TX_ErrorState          (ENABLE := 1, Prio := 6, PG := 0, PF := PGN_TO_PF(dwPGN1_ErrorState),          PS := PGN_TO_PS(dwPGN1_ErrorState),          SRC := ADR(abyCAN1TX_ErrorState),          LEN := 8, RPT := T#0.25S, RESULT => );
CAN1TX_ProcessState        (ENABLE := 1, Prio := 6, PG := 0, PF := PGN_TO_PF(dwPGN1_ProcessState),        PS := PGN_TO_PS(dwPGN1_ProcessState),        SRC := ADR(abyCAN1TX_ProcessState),        LEN := 8, RPT := T#0.05S, RESULT => );

CAN1TX_CoolTempInMin       (ENABLE := 1, Prio := 6, PG := 0, PF := PGN_TO_PF(dwPGN1_CoolTempInMin),       PS := PGN_TO_PS(dwPGN1_CoolTempInMin),       SRC := ADR(abyCAN1TX_CoolTempInMin),       LEN := 8, RPT := T#1S,    RESULT => );

CAN1TX_GN2_Pres            (ENABLE := 1, Prio := 6, PG := 0, PF := PGN_TO_PF(dwPGN1_GN2_Pres),            PS := PGN_TO_PS(dwPGN1_GN2_Pres),            SRC := ADR(abyCAN1TX_GN2_Pres),            LEN := 8, RPT := T#0.5S, RESULT => );
END_PROGRAM

(* POU CAN2_J1939/CAN2_J1939_Transmit_processing, ST *)
PROGRAM CAN2_J1939_Transmit_processing

VAR_INPUT
	bInit               : BOOL;
END_VAR

VAR
	(*dwSignal_DM3_rqst : DWORD := 16#00FECC;(*65228*)*)
	dwSignal_DM2_rqst   : DWORD := 16#00FECB;(*65227*)
	dwSignal_EHR_rqst   : DWORD := 16#00FEE5;(*65253*)
	dwSignal_LFC_rqst   : DWORD := 16#00FEE9;(*65257*)
	dwContentArray      : ARRAY [0..2] OF DWORD;
	dwContent           : DWORD := 0;

	bResetErrorsECU3    : BOOL := 0;(**)

	instMemCpy          : MEMCPY;
	i                   : INT;
END_VAR
(*-----------------------------------------------------------------------------------------------------------------------------------------------------------------------------------*)
(**)

dwContentArray[0] := dwSignal_DM2_rqst;
dwContentArray[1] := dwSignal_EHR_rqst;
dwContentArray[2] := dwSignal_LFC_rqst;

IF bInit = 1 THEN dwContent := dwContentArray[0]; END_IF;

instMemCpy(DST:=ADR(abyCAN2TX_RQST_PGN[1]), SRC:=ADR(dwContent), LEN:=3);

CAN2TX_RQST_PGN((*ENABLE := 1,*) Prio := 6, PG := 0, PF := PGN_TO_PF(dwPGN2_RQST_PGN), PS := PGN_TO_PS(dwPGN2_RQST_PGN), SRC := ADR(abyCAN2TX_RQST_PGN), LEN := 3, RPT := T#0.35S, RESULT => );

IF CAN2TX_RQST_PGN.RESULT = 1
THEN
	IF i <= 2
	THEN
		dwContent := dwContentArray[i];
		i := i + 1;
	ELSE
		i := 0;
	END_IF;
END_IF;

(*-----------------------------------------------------------------------------------------------------------------------------------------------------------------------------------*)
(**)

IF bInit = 1 THEN bResetErrorsECU3 := 1; END_IF;

abyCAN2TX_AC[1] := 16#C8;
abyCAN2TX_AC[2] := 16#3F;
abyCAN2TX_AC[3] := 16#5C;
abyCAN2TX_AC[4] := 16#12;
abyCAN2TX_AC[5] := 16#00;
abyCAN2TX_AC[6] := 16#3C;
abyCAN2TX_AC[7] := 16#00;
abyCAN2TX_AC[8] := 16#80;

IF bResetErrorsECU3 = 1
THEN
	IF CAN2TX_AC.RESULT <> 1
	THEN
		CAN2TX_AC.ENABLE := 1;
	ELSE
		bResetErrorsECU3 := 0;
		CAN2TX_AC.ENABLE := 0;
	END_IF;
END_IF;

CAN2TX_AC((*ENABLE := 1,*) Prio := 6, PG := 0, PF := PGN_TO_PF(dwPGN2_AC), PS := PGN_TO_PS(dwPGN2_AC), SRC := ADR(abyCAN2TX_AC), LEN := 8, RPT := T#1S, RESULT => );

(*-----------------------------------------------------------------------------------------------------------------------------------------------------------------------------------*)
(**)

IF bResetErrorsECU1 = 1
THEN
	IF CAN2TX_DM3.RESULT <> 1
	THEN
		CAN2TX_DM3.ENABLE := 1;
	ELSE
		bResetErrorsECU1 := 0;
		CAN2TX_DM3.ENABLE := 0;
	END_IF;
END_IF;

CAN2TX_DM3((*ENABLE := 1,*) Prio := 6, PG := 0, PF := PGN_TO_PF(dwPGN2_DM3), PS := PGN_TO_PS(dwPGN2_DM3), SRC := ADR(abyCAN2TX_DM3), LEN := 0, RPT := T#1S, RESULT => );

(*-----------------------------------------------------------------------------------------------------------------------------------------------------------------------------------*)
(**)

IF bResetErrorsECU2 = 1
THEN
	IF CAN2TX_DM22.RESULT <> 1
	THEN
		CAN2TX_DM22.ENABLE := 1;
	ELSE
		bResetErrorsECU2 := 0;
		CAN2TX_DM22.ENABLE := 0;
	END_IF;
END_IF;

abyCAN2TX_DM22[1] := 16#01;
abyCAN2TX_DM22[2] := 16#FF;
abyCAN2TX_DM22[3] := 16#FF;
abyCAN2TX_DM22[4] := 16#FF;
abyCAN2TX_DM22[5] := 16#FF;

instMemCpy(DST := ADR(abyCAN2TX_DM22[6]), SRC := ADR(adwErrors_SPN_FMI_DM2[1]), LEN := 3);

CAN2TX_DM22((*ENABLE := 1,*) Prio := 6, PG := 0, PF := PGN_TO_PF(dwPGN2_DM22), PS := PGN_TO_PS(dwPGN2_DM22), SRC := ADR(abyCAN2TX_DM22), LEN := 8, RPT := T#1S, RESULT => );
END_PROGRAM

(* POU Default_Settings/Default_Settings_TestMode_processing, ST *)
PROGRAM Default_Settings_TestMode_processing

VAR_INPUT
	bInit                           : BOOL;
END_VAR

VAR
	DefaultSettingsTestModeRecovery : FLASH_TO_PAGE_CHANNEL;
END_VAR
(*-----------------------------------------------------------------------------------------------------------------------------------------------------------------------------------*)
(*Восстановление заводских установок*)

IF bCurrModeChange = 1 AND dwCurrMode = 0 THEN

(*Channel_00*)
	aPage_Channel[00].PARAM_NAME := 'Channel_00_AIN01';
	aPage_Channel[00].PARAM_00   := 0;
	aPage_Channel[00].PARAM_01   := 3259;
	aPage_Channel[00].PARAM_02   := 648;
	aPage_Channel[00].PARAM_03   := 20;
	aPage_Channel[00].PARAM_04   := 4;
	aPage_Channel[00].PARAM_05   := 100;
	aPage_Channel[00].PARAM_06   := 0;
	aPage_Channel[00].PARAM_07   := 0;
	aPage_Channel[00].PARAM_08   := 0;
	aPage_Channel[00].PARAM_09   := 1;
	aPage_Channel[00].PARAM_10   := 0;

(*Channel_01*)
	aPage_Channel[01].PARAM_NAME := 'Channel_01_AIN02';
	aPage_Channel[01].PARAM_00   := 0;
	aPage_Channel[01].PARAM_01   := 3259;
	aPage_Channel[01].PARAM_02   := 648;
	aPage_Channel[01].PARAM_03   := 20;
	aPage_Channel[01].PARAM_04   := 4;
	aPage_Channel[01].PARAM_05   := 100;
	aPage_Channel[01].PARAM_06   := 0;
	aPage_Channel[01].PARAM_07   := 0;
	aPage_Channel[01].PARAM_08   := 0;
	aPage_Channel[01].PARAM_09   := 2;
	aPage_Channel[01].PARAM_10   := 0;

(*Channel_02*)
	aPage_Channel[02].PARAM_NAME := 'Channel_02_AIN03';
	aPage_Channel[02].PARAM_00   := 0;
	aPage_Channel[02].PARAM_01   := 3259;
	aPage_Channel[02].PARAM_02   := 648;
	aPage_Channel[02].PARAM_03   := 20;
	aPage_Channel[02].PARAM_04   := 4;
	aPage_Channel[02].PARAM_05   := 100;
	aPage_Channel[02].PARAM_06   := 0;
	aPage_Channel[02].PARAM_07   := 0;
	aPage_Channel[02].PARAM_08   := 0;
	aPage_Channel[02].PARAM_09   := 3;
	aPage_Channel[02].PARAM_10   := 0;

(*Channel_03*)
	aPage_Channel[03].PARAM_NAME := 'Channel_03_AIN04';
	aPage_Channel[03].PARAM_00   := 0;
	aPage_Channel[03].PARAM_01   := 3259;
	aPage_Channel[03].PARAM_02   := 648;
	aPage_Channel[03].PARAM_03   := 20;
	aPage_Channel[03].PARAM_04   := 4;
	aPage_Channel[03].PARAM_05   := 100;
	aPage_Channel[03].PARAM_06   := 0;
	aPage_Channel[03].PARAM_07   := 0;
	aPage_Channel[03].PARAM_08   := 0;
	aPage_Channel[03].PARAM_09   := 4;
	aPage_Channel[03].PARAM_10   := 0;

(*Channel_04*)
	aPage_Channel[04].PARAM_NAME := 'Channel_04_AIN05';
	aPage_Channel[04].PARAM_00   := 0;
	aPage_Channel[04].PARAM_01   := 3259;
	aPage_Channel[04].PARAM_02   := 648;
	aPage_Channel[04].PARAM_03   := 20;
	aPage_Channel[04].PARAM_04   := 4;
	aPage_Channel[04].PARAM_05   := 100;
	aPage_Channel[04].PARAM_06   := 0;
	aPage_Channel[04].PARAM_07   := 0;
	aPage_Channel[04].PARAM_08   := 0;
	aPage_Channel[04].PARAM_09   := 5;
	aPage_Channel[04].PARAM_10   := 0;

(*Channel_05*)
	aPage_Channel[05].PARAM_NAME := 'Channel_05_AIN06';
	aPage_Channel[05].PARAM_00   := 0;
	aPage_Channel[05].PARAM_01   := 3259;
	aPage_Channel[05].PARAM_02   := 648;
	aPage_Channel[05].PARAM_03   := 20;
	aPage_Channel[05].PARAM_04   := 4;
	aPage_Channel[05].PARAM_05   := 100;
	aPage_Channel[05].PARAM_06   := 0;
	aPage_Channel[05].PARAM_07   := 0;
	aPage_Channel[05].PARAM_08   := 0;
	aPage_Channel[05].PARAM_09   := 6;
	aPage_Channel[05].PARAM_10   := 0;

(*Channel_06*)
	aPage_Channel[06].PARAM_NAME := 'Channel_06_AIN07';
	aPage_Channel[06].PARAM_00   := 0;
	aPage_Channel[06].PARAM_01   := 3259;
	aPage_Channel[06].PARAM_02   := 648;
	aPage_Channel[06].PARAM_03   := 20;
	aPage_Channel[06].PARAM_04   := 4;
	aPage_Channel[06].PARAM_05   := 100;
	aPage_Channel[06].PARAM_06   := 0;
	aPage_Channel[06].PARAM_07   := 0;
	aPage_Channel[06].PARAM_08   := 0;
	aPage_Channel[06].PARAM_09   := 7;
	aPage_Channel[06].PARAM_10   := 0;

(*Channel_07*)
	aPage_Channel[07].PARAM_NAME := 'Channel_07_AIN08';
	aPage_Channel[07].PARAM_00   := 0;
	aPage_Channel[07].PARAM_01   := 3259;
	aPage_Channel[07].PARAM_02   := 648;
	aPage_Channel[07].PARAM_03   := 20;
	aPage_Channel[07].PARAM_04   := 4;
	aPage_Channel[07].PARAM_05   := 100;
	aPage_Channel[07].PARAM_06   := 0;
	aPage_Channel[07].PARAM_07   := 0;
	aPage_Channel[07].PARAM_08   := 0;
	aPage_Channel[07].PARAM_09   := 8;
	aPage_Channel[07].PARAM_10   := 0;

(*Channel_08*)
	aPage_Channel[08].PARAM_NAME := 'Channel_08_AIN09';
	aPage_Channel[08].PARAM_00   := 0;
	aPage_Channel[08].PARAM_01   := 3259;
	aPage_Channel[08].PARAM_02   := 648;
	aPage_Channel[08].PARAM_03   := 20;
	aPage_Channel[08].PARAM_04   := 4;
	aPage_Channel[08].PARAM_05   := 100;
	aPage_Channel[08].PARAM_06   := 0;
	aPage_Channel[08].PARAM_07   := 0;
	aPage_Channel[08].PARAM_08   := 0;
	aPage_Channel[08].PARAM_09   := 9;
	aPage_Channel[08].PARAM_10   := 0;

(*Channel_09*)
	aPage_Channel[09].PARAM_NAME := 'Channel_09_AIN10';
	aPage_Channel[09].PARAM_00   := 0;
	aPage_Channel[09].PARAM_01   := 3259;
	aPage_Channel[09].PARAM_02   := 648;
	aPage_Channel[09].PARAM_03   := 20;
	aPage_Channel[09].PARAM_04   := 4;
	aPage_Channel[09].PARAM_05   := 100;
	aPage_Channel[09].PARAM_06   := 0;
	aPage_Channel[09].PARAM_07   := 0;
	aPage_Channel[09].PARAM_08   := 0;
	aPage_Channel[09].PARAM_09   := 10;
	aPage_Channel[09].PARAM_10   := 0;

(*Channel_10*)
	aPage_Channel[10].PARAM_NAME := 'Channel_10_AIN11';
	aPage_Channel[10].PARAM_00   := 0;
	aPage_Channel[10].PARAM_01   := 3259;
	aPage_Channel[10].PARAM_02   := 648;
	aPage_Channel[10].PARAM_03   := 20;
	aPage_Channel[10].PARAM_04   := 4;
	aPage_Channel[10].PARAM_05   := 100;
	aPage_Channel[10].PARAM_06   := 0;
	aPage_Channel[10].PARAM_07   := 0;
	aPage_Channel[10].PARAM_08   := 0;
	aPage_Channel[10].PARAM_09   := 11;
	aPage_Channel[10].PARAM_10   := 0;

(*Channel_11*)
	aPage_Channel[11].PARAM_NAME := 'Channel_11_AIN12';
	aPage_Channel[11].PARAM_00   := 0;
	aPage_Channel[11].PARAM_01   := 3259;
	aPage_Channel[11].PARAM_02   := 648;
	aPage_Channel[11].PARAM_03   := 20;
	aPage_Channel[11].PARAM_04   := 4;
	aPage_Channel[11].PARAM_05   := 100;
	aPage_Channel[11].PARAM_06   := 0;
	aPage_Channel[11].PARAM_07   := 0;
	aPage_Channel[11].PARAM_08   := 0;
	aPage_Channel[11].PARAM_09   := 12;
	aPage_Channel[11].PARAM_10   := 0;

(*Channel_12*)
	aPage_Channel[12].PARAM_NAME := 'Channel_12_AIN13';
	aPage_Channel[12].PARAM_00   := 0;
	aPage_Channel[12].PARAM_01   := 3259;
	aPage_Channel[12].PARAM_02   := 648;
	aPage_Channel[12].PARAM_03   := 20;
	aPage_Channel[12].PARAM_04   := 4;
	aPage_Channel[12].PARAM_05   := 100;
	aPage_Channel[12].PARAM_06   := 0;
	aPage_Channel[12].PARAM_07   := 0;
	aPage_Channel[12].PARAM_08   := 0;
	aPage_Channel[12].PARAM_09   := 13;
	aPage_Channel[12].PARAM_10   := 0;

(*Channel_13*)
	aPage_Channel[13].PARAM_NAME := 'Channel_13_AIN14';
	aPage_Channel[13].PARAM_00   := 0;
	aPage_Channel[13].PARAM_01   := 3259;
	aPage_Channel[13].PARAM_02   := 648;
	aPage_Channel[13].PARAM_03   := 20;
	aPage_Channel[13].PARAM_04   := 4;
	aPage_Channel[13].PARAM_05   := 100;
	aPage_Channel[13].PARAM_06   := 0;
	aPage_Channel[13].PARAM_07   := 0;
	aPage_Channel[13].PARAM_08   := 0;
	aPage_Channel[13].PARAM_09   := 14;
	aPage_Channel[13].PARAM_10   := 0;

(*Channel_14*)
	aPage_Channel[14].PARAM_NAME := 'Channel_14_AIN15';
	aPage_Channel[14].PARAM_00   := 0;
	aPage_Channel[14].PARAM_01   := 3259;
	aPage_Channel[14].PARAM_02   := 648;
	aPage_Channel[14].PARAM_03   := 20;
	aPage_Channel[14].PARAM_04   := 4;
	aPage_Channel[14].PARAM_05   := 100;
	aPage_Channel[14].PARAM_06   := 0;
	aPage_Channel[14].PARAM_07   := 0;
	aPage_Channel[14].PARAM_08   := 0;
	aPage_Channel[14].PARAM_09   := 15;
	aPage_Channel[14].PARAM_10   := 0;

(*Channel_15*)
	aPage_Channel[15].PARAM_NAME := 'Channel_15_AIN16';
	aPage_Channel[15].PARAM_00   := 0;
	aPage_Channel[15].PARAM_01   := 3259;
	aPage_Channel[15].PARAM_02   := 648;
	aPage_Channel[15].PARAM_03   := 20;
	aPage_Channel[15].PARAM_04   := 4;
	aPage_Channel[15].PARAM_05   := 100;
	aPage_Channel[15].PARAM_06   := 0;
	aPage_Channel[15].PARAM_07   := 0;
	aPage_Channel[15].PARAM_08   := 0;
	aPage_Channel[15].PARAM_09   := 16;
	aPage_Channel[15].PARAM_10   := 0;

(*Channel_16*)
	aPage_Channel[16].PARAM_NAME := 'Channel_16_PIN01';
	aPage_Channel[16].PARAM_00   := 1;
	aPage_Channel[16].PARAM_01   := 10_000;
	aPage_Channel[16].PARAM_02   := 0;
	aPage_Channel[16].PARAM_03   := 100;
	aPage_Channel[16].PARAM_04   := 0;
	aPage_Channel[16].PARAM_05   := 1_000;
	aPage_Channel[16].PARAM_06   := 0;
	aPage_Channel[16].PARAM_07   := 0;
	aPage_Channel[16].PARAM_08   := 0;
	aPage_Channel[16].PARAM_09   := 1;
	aPage_Channel[16].PARAM_10   := 0;

(*Channel_17*)
	aPage_Channel[17].PARAM_NAME := 'Channel_17_PIN02';
	aPage_Channel[17].PARAM_00   := 1;
	aPage_Channel[17].PARAM_01   := 10_000;
	aPage_Channel[17].PARAM_02   := 0;
	aPage_Channel[17].PARAM_03   := 100;
	aPage_Channel[17].PARAM_04   := 0;
	aPage_Channel[17].PARAM_05   := 1_000;
	aPage_Channel[17].PARAM_06   := 0;
	aPage_Channel[17].PARAM_07   := 0;
	aPage_Channel[17].PARAM_08   := 0;
	aPage_Channel[17].PARAM_09   := 2;
	aPage_Channel[17].PARAM_10   := 0;

(*Channel_18*)
	aPage_Channel[18].PARAM_NAME := 'Channel_18_PIN03';
	aPage_Channel[18].PARAM_00   := 1;
	aPage_Channel[18].PARAM_01   := 10_000;
	aPage_Channel[18].PARAM_02   := 0;
	aPage_Channel[18].PARAM_03   := 100;
	aPage_Channel[18].PARAM_04   := 0;
	aPage_Channel[18].PARAM_05   := 1_000;
	aPage_Channel[18].PARAM_06   := 0;
	aPage_Channel[18].PARAM_07   := 0;
	aPage_Channel[18].PARAM_08   := 0;
	aPage_Channel[18].PARAM_09   := 3;
	aPage_Channel[18].PARAM_10   := 0;

(*Channel_19*)
	aPage_Channel[19].PARAM_NAME := 'Channel_19_PIN04';
	aPage_Channel[19].PARAM_00   := 1;
	aPage_Channel[19].PARAM_01   := 10_000;
	aPage_Channel[19].PARAM_02   := 0;
	aPage_Channel[19].PARAM_03   := 100;
	aPage_Channel[19].PARAM_04   := 0;
	aPage_Channel[19].PARAM_05   := 1_000;
	aPage_Channel[19].PARAM_06   := 0;
	aPage_Channel[19].PARAM_07   := 0;
	aPage_Channel[19].PARAM_08   := 0;
	aPage_Channel[19].PARAM_09   := 4;
	aPage_Channel[19].PARAM_10   := 0;

(*Channel_20*)
	aPage_Channel[20].PARAM_NAME := 'Channel_20_PIN05';
	aPage_Channel[20].PARAM_00   := 1;
	aPage_Channel[20].PARAM_01   := 10_000;
	aPage_Channel[20].PARAM_02   := 0;
	aPage_Channel[20].PARAM_03   := 100;
	aPage_Channel[20].PARAM_04   := 0;
	aPage_Channel[20].PARAM_05   := 1_000;
	aPage_Channel[20].PARAM_06   := 0;
	aPage_Channel[20].PARAM_07   := 0;
	aPage_Channel[20].PARAM_08   := 0;
	aPage_Channel[20].PARAM_09   := 5;
	aPage_Channel[20].PARAM_10   := 0;

(*Channel_21*)
	aPage_Channel[21].PARAM_NAME := 'Channel_21_PIN06';
	aPage_Channel[21].PARAM_00   := 1;
	aPage_Channel[21].PARAM_01   := 10_000;
	aPage_Channel[21].PARAM_02   := 0;
	aPage_Channel[21].PARAM_03   := 100;
	aPage_Channel[21].PARAM_04   := 0;
	aPage_Channel[21].PARAM_05   := 1_000;
	aPage_Channel[21].PARAM_06   := 0;
	aPage_Channel[21].PARAM_07   := 0;
	aPage_Channel[21].PARAM_08   := 0;
	aPage_Channel[21].PARAM_09   := 6;
	aPage_Channel[21].PARAM_10   := 0;

(*Channel_22*)
	aPage_Channel[22].PARAM_NAME := 'Channel_22_PIN07';
	aPage_Channel[22].PARAM_00   := 1;
	aPage_Channel[22].PARAM_01   := 10_000;
	aPage_Channel[22].PARAM_02   := 0;
	aPage_Channel[22].PARAM_03   := 100;
	aPage_Channel[22].PARAM_04   := 0;
	aPage_Channel[22].PARAM_05   := 1_000;
	aPage_Channel[22].PARAM_06   := 0;
	aPage_Channel[22].PARAM_07   := 0;
	aPage_Channel[22].PARAM_08   := 0;
	aPage_Channel[22].PARAM_09   := 7;
	aPage_Channel[22].PARAM_10   := 0;

(*Channel_23*)
	aPage_Channel[23].PARAM_NAME := 'Channel_23_PIN08';
	aPage_Channel[23].PARAM_00   := 1;
	aPage_Channel[23].PARAM_01   := 10_000;
	aPage_Channel[23].PARAM_02   := 0;
	aPage_Channel[23].PARAM_03   := 100;
	aPage_Channel[23].PARAM_04   := 0;
	aPage_Channel[23].PARAM_05   := 1_000;
	aPage_Channel[23].PARAM_06   := 0;
	aPage_Channel[23].PARAM_07   := 0;
	aPage_Channel[23].PARAM_08   := 0;
	aPage_Channel[23].PARAM_09   := 8;
	aPage_Channel[23].PARAM_10   := 0;

(*Channel_24*)
	aPage_Channel[24].PARAM_NAME := 'Channel_24_PWM01';
	aPage_Channel[24].PARAM_00   := 2;
	aPage_Channel[24].PARAM_01   := 100;
	aPage_Channel[24].PARAM_02   := 0;
	aPage_Channel[24].PARAM_03   := 100;
	aPage_Channel[24].PARAM_04   := 0;
	aPage_Channel[24].PARAM_05   := 4_000;
	aPage_Channel[24].PARAM_06   := 0;
	aPage_Channel[24].PARAM_07   := 0;
	aPage_Channel[24].PARAM_08   := 0;
	aPage_Channel[24].PARAM_09   := 1;
	aPage_Channel[24].PARAM_10   := 0;

(*Channel_25*)
	aPage_Channel[25].PARAM_NAME := 'Channel_25_PWM02';
	aPage_Channel[25].PARAM_00   := 2;
	aPage_Channel[25].PARAM_01   := 100;
	aPage_Channel[25].PARAM_02   := 0;
	aPage_Channel[25].PARAM_03   := 100;
	aPage_Channel[25].PARAM_04   := 0;
	aPage_Channel[25].PARAM_05   := 4_000;
	aPage_Channel[25].PARAM_06   := 0;
	aPage_Channel[25].PARAM_07   := 0;
	aPage_Channel[25].PARAM_08   := 0;
	aPage_Channel[25].PARAM_09   := 2;
	aPage_Channel[25].PARAM_10   := 0;

(*Channel_26*)
	aPage_Channel[26].PARAM_NAME := 'Channel_26_PWM03';
	aPage_Channel[26].PARAM_00   := 2;
	aPage_Channel[26].PARAM_01   := 100;
	aPage_Channel[26].PARAM_02   := 0;
	aPage_Channel[26].PARAM_03   := 100;
	aPage_Channel[26].PARAM_04   := 0;
	aPage_Channel[26].PARAM_05   := 4_000;
	aPage_Channel[26].PARAM_06   := 0;
	aPage_Channel[26].PARAM_07   := 0;
	aPage_Channel[26].PARAM_08   := 0;
	aPage_Channel[26].PARAM_09   := 3;
	aPage_Channel[26].PARAM_10   := 0;

(*Channel_27*)
	aPage_Channel[27].PARAM_NAME := 'Channel_27_PWM04';
	aPage_Channel[27].PARAM_00   := 2;
	aPage_Channel[27].PARAM_01   := 100;
	aPage_Channel[27].PARAM_02   := 0;
	aPage_Channel[27].PARAM_03   := 100;
	aPage_Channel[27].PARAM_04   := 0;
	aPage_Channel[27].PARAM_05   := 4_000;
	aPage_Channel[27].PARAM_06   := 0;
	aPage_Channel[27].PARAM_07   := 0;
	aPage_Channel[27].PARAM_08   := 0;
	aPage_Channel[27].PARAM_09   := 4;
	aPage_Channel[27].PARAM_10   := 0;

(*Channel_28*)
	aPage_Channel[28].PARAM_NAME := 'Channel_28_PWM05';
	aPage_Channel[28].PARAM_00   := 2;
	aPage_Channel[28].PARAM_01   := 100;
	aPage_Channel[28].PARAM_02   := 0;
	aPage_Channel[28].PARAM_03   := 100;
	aPage_Channel[28].PARAM_04   := 0;
	aPage_Channel[28].PARAM_05   := 4_000;
	aPage_Channel[28].PARAM_06   := 0;
	aPage_Channel[28].PARAM_07   := 0;
	aPage_Channel[28].PARAM_08   := 0;
	aPage_Channel[28].PARAM_09   := 5;
	aPage_Channel[28].PARAM_10   := 0;

(*Channel_29*)
	aPage_Channel[29].PARAM_NAME := 'Channel_29_PWM06';
	aPage_Channel[29].PARAM_00   := 2;
	aPage_Channel[29].PARAM_01   := 100;
	aPage_Channel[29].PARAM_02   := 0;
	aPage_Channel[29].PARAM_03   := 100;
	aPage_Channel[29].PARAM_04   := 0;
	aPage_Channel[29].PARAM_05   := 4_000;
	aPage_Channel[29].PARAM_06   := 0;
	aPage_Channel[29].PARAM_07   := 0;
	aPage_Channel[29].PARAM_08   := 0;
	aPage_Channel[29].PARAM_09   := 6;
	aPage_Channel[29].PARAM_10   := 0;

(*Channel_30*)
	aPage_Channel[30].PARAM_NAME := 'Channel_30_PWM07';
	aPage_Channel[30].PARAM_00   := 2;
	aPage_Channel[30].PARAM_01   := 100;
	aPage_Channel[30].PARAM_02   := 0;
	aPage_Channel[30].PARAM_03   := 100;
	aPage_Channel[30].PARAM_04   := 0;
	aPage_Channel[30].PARAM_05   := 4_000;
	aPage_Channel[30].PARAM_06   := 0;
	aPage_Channel[30].PARAM_07   := 0;
	aPage_Channel[30].PARAM_08   := 0;
	aPage_Channel[30].PARAM_09   := 7;
	aPage_Channel[30].PARAM_10   := 0;

(*Channel_31*)
	aPage_Channel[31].PARAM_NAME := 'Channel_31_PWM08';
	aPage_Channel[31].PARAM_00   := 2;
	aPage_Channel[31].PARAM_01   := 100;
	aPage_Channel[31].PARAM_02   := 0;
	aPage_Channel[31].PARAM_03   := 100;
	aPage_Channel[31].PARAM_04   := 0;
	aPage_Channel[31].PARAM_05   := 4_000;
	aPage_Channel[31].PARAM_06   := 0;
	aPage_Channel[31].PARAM_07   := 0;
	aPage_Channel[31].PARAM_08   := 0;
	aPage_Channel[31].PARAM_09   := 8;
	aPage_Channel[31].PARAM_10   := 0;

(*Channel_32*)
	aPage_Channel[32].PARAM_NAME := 'Channel_32_PID01';
	aPage_Channel[32].PARAM_00   := 3;
	aPage_Channel[32].PARAM_01   := 50;
	aPage_Channel[32].PARAM_02   := 30;
	aPage_Channel[32].PARAM_03   := 5;
	aPage_Channel[32].PARAM_04   := 0;
	aPage_Channel[32].PARAM_05   := 1;
	aPage_Channel[32].PARAM_06   := 0;
	aPage_Channel[32].PARAM_07   := 0;
	aPage_Channel[32].PARAM_08   := 0;
	aPage_Channel[32].PARAM_09   := 1;
	aPage_Channel[32].PARAM_10   := 0;

(*Channel_33*)
	aPage_Channel[33].PARAM_NAME := 'Channel_33_PID02';
	aPage_Channel[33].PARAM_00   := 3;
	aPage_Channel[33].PARAM_01   := 50;
	aPage_Channel[33].PARAM_02   := 30;
	aPage_Channel[33].PARAM_03   := 5;
	aPage_Channel[33].PARAM_04   := 0;
	aPage_Channel[33].PARAM_05   := 1;
	aPage_Channel[33].PARAM_06   := 0;
	aPage_Channel[33].PARAM_07   := 0;
	aPage_Channel[33].PARAM_08   := 0;
	aPage_Channel[33].PARAM_09   := 2;
	aPage_Channel[33].PARAM_10   := 0;

(*Channel_34*)
	aPage_Channel[34].PARAM_NAME := 'Channel_34_PID03';
	aPage_Channel[34].PARAM_00   := 3;
	aPage_Channel[34].PARAM_01   := 50;
	aPage_Channel[34].PARAM_02   := 30;
	aPage_Channel[34].PARAM_03   := 5;
	aPage_Channel[34].PARAM_04   := 0;
	aPage_Channel[34].PARAM_05   := 1;
	aPage_Channel[34].PARAM_06   := 0;
	aPage_Channel[34].PARAM_07   := 0;
	aPage_Channel[34].PARAM_08   := 0;
	aPage_Channel[34].PARAM_09   := 3;
	aPage_Channel[34].PARAM_10   := 0;

(*Channel_35*)
	aPage_Channel[35].PARAM_NAME := 'Channel_35_PID04';
	aPage_Channel[35].PARAM_00   := 3;
	aPage_Channel[35].PARAM_01   := 50;
	aPage_Channel[35].PARAM_02   := 30;
	aPage_Channel[35].PARAM_03   := 5;
	aPage_Channel[35].PARAM_04   := 0;
	aPage_Channel[35].PARAM_05   := 1;
	aPage_Channel[35].PARAM_06   := 0;
	aPage_Channel[35].PARAM_07   := 0;
	aPage_Channel[35].PARAM_08   := 0;
	aPage_Channel[35].PARAM_09   := 4;
	aPage_Channel[35].PARAM_10   := 0;

(*Channel_36*)
	aPage_Channel[36].PARAM_NAME := 'Channel_36_PID05';
	aPage_Channel[36].PARAM_00   := 3;
	aPage_Channel[36].PARAM_01   := 50;
	aPage_Channel[36].PARAM_02   := 30;
	aPage_Channel[36].PARAM_03   := 5;
	aPage_Channel[36].PARAM_04   := 0;
	aPage_Channel[36].PARAM_05   := 1;
	aPage_Channel[36].PARAM_06   := 0;
	aPage_Channel[36].PARAM_07   := 0;
	aPage_Channel[36].PARAM_08   := 0;
	aPage_Channel[36].PARAM_09   := 5;
	aPage_Channel[36].PARAM_10   := 0;

(*Channel_37*)
	aPage_Channel[37].PARAM_NAME := 'Channel_37_PID06';
	aPage_Channel[37].PARAM_00   := 3;
	aPage_Channel[37].PARAM_01   := 50;
	aPage_Channel[37].PARAM_02   := 30;
	aPage_Channel[37].PARAM_03   := 5;
	aPage_Channel[37].PARAM_04   := 0;
	aPage_Channel[37].PARAM_05   := 1;
	aPage_Channel[37].PARAM_06   := 0;
	aPage_Channel[37].PARAM_07   := 0;
	aPage_Channel[37].PARAM_08   := 0;
	aPage_Channel[37].PARAM_09   := 6;
	aPage_Channel[37].PARAM_10   := 0;

(*Channel_38*)
	aPage_Channel[38].PARAM_NAME := 'Channel_38_PID07';
	aPage_Channel[38].PARAM_00   := 3;
	aPage_Channel[38].PARAM_01   := 50;
	aPage_Channel[38].PARAM_02   := 30;
	aPage_Channel[38].PARAM_03   := 5;
	aPage_Channel[38].PARAM_04   := 0;
	aPage_Channel[38].PARAM_05   := 1;
	aPage_Channel[38].PARAM_06   := 0;
	aPage_Channel[38].PARAM_07   := 0;
	aPage_Channel[38].PARAM_08   := 0;
	aPage_Channel[38].PARAM_09   := 7;
	aPage_Channel[38].PARAM_10   := 0;

(*Channel_39*)
	aPage_Channel[39].PARAM_NAME := 'Channel_39_PID08';
	aPage_Channel[39].PARAM_00   := 3;
	aPage_Channel[39].PARAM_01   := 50;
	aPage_Channel[39].PARAM_02   := 30;
	aPage_Channel[39].PARAM_03   := 5;
	aPage_Channel[39].PARAM_04   := 0;
	aPage_Channel[39].PARAM_05   := 1;
	aPage_Channel[39].PARAM_06   := 0;
	aPage_Channel[39].PARAM_07   := 0;
	aPage_Channel[39].PARAM_08   := 0;
	aPage_Channel[39].PARAM_09   := 8;
	aPage_Channel[39].PARAM_10   := 0;

(*Channel_40*)
	aPage_Channel[40].PARAM_NAME := 'Channel_40_ENC01';
	aPage_Channel[40].PARAM_00   := 4;
	aPage_Channel[40].PARAM_01   := 100;
	aPage_Channel[40].PARAM_02   := 0;
	aPage_Channel[40].PARAM_03   := 0;
	aPage_Channel[40].PARAM_04   := 0;
	aPage_Channel[40].PARAM_05   := 0;
	aPage_Channel[40].PARAM_06   := 0;
	aPage_Channel[40].PARAM_07   := 0;
	aPage_Channel[40].PARAM_08   := 0;
	aPage_Channel[40].PARAM_09   := 1;
	aPage_Channel[40].PARAM_10   := 0;

(*Channel_41*)
	aPage_Channel[41].PARAM_NAME := 'Channel_41_ENC02';
	aPage_Channel[41].PARAM_00   := 4;
	aPage_Channel[41].PARAM_01   := 200;
	aPage_Channel[41].PARAM_02   := 0;
	aPage_Channel[41].PARAM_03   := 0;
	aPage_Channel[41].PARAM_04   := 0;
	aPage_Channel[41].PARAM_05   := 0;
	aPage_Channel[41].PARAM_06   := 0;
	aPage_Channel[41].PARAM_07   := 0;
	aPage_Channel[41].PARAM_08   := 0;
	aPage_Channel[41].PARAM_09   := 2;
	aPage_Channel[41].PARAM_10   := 0;

(*Channel_42*)
	aPage_Channel[42].PARAM_NAME := 'Channel_42_ENC03';
	aPage_Channel[42].PARAM_00   := 4;
	aPage_Channel[42].PARAM_01   := 300;
	aPage_Channel[42].PARAM_02   := 0;
	aPage_Channel[42].PARAM_03   := 0;
	aPage_Channel[42].PARAM_04   := 0;
	aPage_Channel[42].PARAM_05   := 0;
	aPage_Channel[42].PARAM_06   := 0;
	aPage_Channel[42].PARAM_07   := 0;
	aPage_Channel[42].PARAM_08   := 0;
	aPage_Channel[42].PARAM_09   := 3;
	aPage_Channel[42].PARAM_10   := 0;

